KUKA KRL program: EPS_2_251191_MH01A_A_20251103013754.src

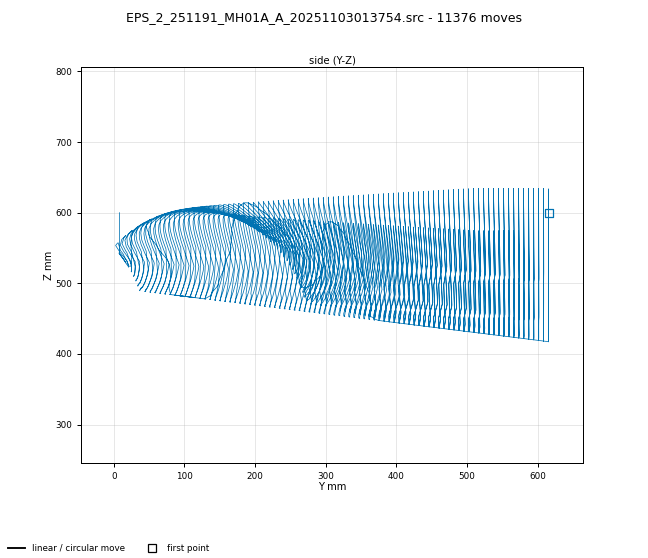
[picture p0: tool path of EPS_2_251191_MH01A_A_20251103013754.src, 11376 of 11378 moves have a stored position in this frame; points joined in program order, loops and branches not executed]
&ACCESS RVP
&REL 4
&COMMENT QRS 19112012
&PARAM EDITMASK = *
DEF PART()
EXT BAS (BAS_COMMAND :IN,REAL :IN )
INT I
BAS (#INITMOV,0 )

;KUKA QRS Post kuka4.cps  Date:22-06-2017 !

File_ID=2898

QRS_PRE_INIT()

;Init var - Until changes are made in qrs_pre_init
Outlet_Square_prg=0
Inlet_1_Square_prg=0
Inlet_2_Square_prg=0
Inlet_3_Square_prg=0
Inlet_4_Square_prg=0
Inlet_5_Square_prg=0

Outlet_1={X 0.000, Y 509.470, Z 509.000, B 0.000, E1 0.000 }
Inlet_1={X 0.000, Y 513.890, Z 449.000, B 0.000, E1 252.000 }
Outlet_1_type=251
Inlet_1_type=251
;QRS#1=Sidecore dimensions
;QRS#2=250-10" PVC SDR 35
;QRS#3=250-10" PVC SDR 35
;QRS#4=
;QRS#5=
;QRS#6=
;QRS#7=
;QRS#8=
;QRS#9=14M PSX
;QRS#10=14M PSX
;QRS#11=
;QRS#12=
;QRS#13=
;QRS#14=
;QRS#15=
;QRS#16=1220x127x914 3'
;QRS#17=EPS Height
;QRS#18=634,5
;QRS#19=*
;QRS#20= UPDATED VERSION 22-06-2017
;QRS#21=*
Outlet_Square=0100
Inlet_1_Square=0100
Inlet_2_Square=0
Inlet_3_Square=0
Inlet_4_Square=0
Inlet_5_Square=0
Mill_Square=1
Outlet_Square_Prg=205
Inlet_1_Square_prg=205

QRS_INIT()

$ADVANCE=5

; T1
PTP {E1 173.596,E2 173.596}
PTP {X 0,Y 615.507,A -85,B 0,C 180,E1 173.596,E2 173.596,E3 0,E4 0,E5 0,E6 0}
QRS_SPEED_INIT()
LIN {X 0,Y 615.507,Z 600,A -85,B 0,C 180,E1 173.596,E2 173.596,E3 0,E4 0,E5 0,E6 0} C_VEL
LIN {X 0,Y 615.507,Z 427.495,A -85,B 0,C 180,E1 173.596,E2 173.596} C_VEL
LIN {X 0,Y 615.507,Z 419.317,A -85,B 0,C 180,E1 173.596,E2 173.596} C_VEL
LIN {X 0,Y 615.493,Z 417.317,A -85,B 0,C 180,E1 173.409,E2 173.409} C_VEL
LIN {X 0,Y 615.481,Z 417.32,A -85,B 0,C 180,E1 170.801,E2 170.801} C_VEL
LIN {X 0,Y 615.475,Z 417.322,A -85,B 0,C 180,E1 168.139,E2 168.139} C_VEL
LIN {X 0,Y 615.49,Z 417.319,A -85,B 0,C 180,E1 165.451,E2 165.451} C_VEL
LIN {X 0,Y 615.49,Z 417.319,A -85,B 0,C 180,E1 162.729,E2 162.729} C_VEL
LIN {X 0,Y 615.486,Z 417.32,A -85,B 0,C 180,E1 159.967,E2 159.967} C_VEL
LIN {X 0,Y 615.477,Z 417.321,A -85,B 0,C 180,E1 157.155,E2 157.155} C_VEL
LIN {X 0,Y 615.484,Z 417.32,A -85,B 0,C 180,E1 154.43,E2 154.43} C_VEL
LIN {X 0,Y 615.492,Z 417.317,A -85,B 0,C 180,E1 151.547,E2 151.547} C_VEL
LIN {X 0,Y 615.483,Z 417.32,A -85,B 0,C 180,E1 148.913,E2 148.913} C_VEL
LIN {X 0,Y 615.486,Z 417.323,A -85,B 0,C 180,E1 146.465,E2 146.465} C_VEL
LIN {X 0,Y 615.488,Z 417.32,A -85,B 0,C 180,E1 143.575,E2 143.575} C_VEL
LIN {X 0,Y 615.484,Z 417.323,A -85,B 0,C 180,E1 140.937,E2 140.937} C_VEL
LIN {X 0,Y 615.487,Z 417.325,A -85,B 0,C 180,E1 138.526,E2 138.526} C_VEL
LIN {X 0,Y 615.491,Z 417.323,A -85,B 0,C 180,E1 135.85,E2 135.85} C_VEL
LIN {X 0,Y 615.492,Z 417.324,A -85,B 0,C 180,E1 133.047,E2 133.047} C_VEL
LIN {X 0,Y 615.497,Z 417.323,A -85,B 0,C 180,E1 130.09,E2 130.09} C_VEL
LIN {X 0,Y 615.484,Z 417.324,A -85,B 0,C 180,E1 127.242,E2 127.242} C_VEL
LIN {X 0,Y 615.496,Z 417.325,A -85,B 0,C 180,E1 124.701,E2 124.701} C_VEL
LIN {X 0,Y 615.48,Z 417.321,A -85,B 0,C 180,E1 122.329,E2 122.329} C_VEL
LIN {X 0,Y 615.498,Z 417.316,A -85,B 0,C 180,E1 119.796,E2 119.796} C_VEL
LIN {X 0,Y 615.486,Z 417.318,A -85,B 0,C 180,E1 117.044,E2 117.044} C_VEL
LIN {X 0,Y 615.478,Z 417.32,A -85,B 0,C 180,E1 114.272,E2 114.272} C_VEL
LIN {X 0,Y 615.479,Z 417.321,A -85,B 0,C 180,E1 111.432,E2 111.432} C_VEL
LIN {X 0,Y 615.481,Z 417.321,A -85,B 0,C 180,E1 108.602,E2 108.602} C_VEL
LIN {X 0,Y 615.491,Z 417.318,A -85,B 0,C 180,E1 105.905,E2 105.905} C_VEL
LIN {X 0,Y 615.48,Z 417.32,A -85,B 0,C 180,E1 103.201,E2 103.201} C_VEL
LIN {X 0,Y 615.478,Z 417.32,A -85,B 0,C 180,E1 100.527,E2 100.527} C_VEL
LIN {X 0,Y 615.489,Z 417.317,A -85,B 0,C 180,E1 97.875,E2 97.875} C_VEL
LIN {X 0,Y 615.484,Z 417.319,A -85,B 0,C 180,E1 95.241,E2 95.241} C_VEL
LIN {X 0,Y 615.478,Z 417.321,A -85,B 0,C 180,E1 92.618,E2 92.618} C_VEL
LIN {X 0,Y 615.491,Z 417.32,A -85,B 0,C 180,E1 90,E2 90} C_VEL
LIN {X 0,Y 615.484,Z 417.324,A -85,B 0,C 180,E1 87.382,E2 87.382} C_VEL
LIN {X 0,Y 615.493,Z 417.325,A -85,B 0,C 180,E1 84.759,E2 84.759} C_VEL
LIN {X 0,Y 615.487,Z 417.327,A -85,B 0,C 180,E1 82.125,E2 82.125} C_VEL
LIN {X 0,Y 615.488,Z 417.324,A -85,B 0,C 180,E1 79.473,E2 79.473} C_VEL
LIN {X 0,Y 615.482,Z 417.324,A -85,B 0,C 180,E1 76.799,E2 76.799} C_VEL
LIN {X 0,Y 615.491,Z 417.321,A -85,B 0,C 180,E1 74.095,E2 74.095} C_VEL
LIN {X 0,Y 615.483,Z 417.323,A -85,B 0,C 180,E1 71.354,E2 71.354} C_VEL
LIN {X 0,Y 615.482,Z 417.324,A -85,B 0,C 180,E1 68.568,E2 68.568} C_VEL
LIN {X 0,Y 615.495,Z 417.323,A -85,B 0,C 180,E1 65.729,E2 65.729} C_VEL
LIN {X 0,Y 615.486,Z 417.328,A -85,B 0,C 180,E1 62.823,E2 62.823} C_VEL
LIN {X 0,Y 615.497,Z 417.323,A -85,B 0,C 180,E1 60.205,E2 60.205} C_VEL
LIN {X 0,Y 615.488,Z 417.323,A -85,B 0,C 180,E1 57.543,E2 57.543} C_VEL
LIN {X 0,Y 615.496,Z 417.434,A -85,B 0,C 180,E1 55.979,E2 55.979} C_VEL
LIN {X 0,Y 615.483,Z 420.003,A -85,B 0,C 180,E1 53.576,E2 53.576} C_VEL
LIN {X 0,Y 615.485,Z 422.805,A -85,B 0,C 180,E1 50.939,E2 50.939} C_VEL
LIN {X 0,Y 615.495,Z 425.526,A -85,B 0,C 180,E1 48.528,E2 48.528} C_VEL
LIN {X 0,Y 615.478,Z 428.644,A -85,B 0,C 180,E1 45.851,E2 45.851} C_VEL
LIN {X 0,Y 615.493,Z 431.993,A -85,B 0,C 180,E1 43.049,E2 43.049} C_VEL
LIN {X 0,Y 615.486,Z 435.606,A -85,B 0,C 180,E1 40.09,E2 40.09} C_VEL
LIN {X 0,Y 615.491,Z 439.16,A -85,B 0,C 180,E1 37.242,E2 37.242} C_VEL
LIN {X 0,Y 615.478,Z 442.382,A -85,B 0,C 180,E1 34.701,E2 34.701} C_VEL
LIN {X 0,Y 615.494,Z 445.903,A -85,B 0,C 180,E1 31.968,E2 31.968} C_VEL
LIN {X 0,Y 615.485,Z 463.146,A -85,B 0,C 180,E1 31.611,E2 31.611} C_VEL
LIN {X 0,Y 615.49,Z 476.555,A -85,B 0,C 180,E1 31.199,E2 31.199} C_VEL
LIN {X 0,Y 615.481,Z 490.214,A -85,B 0,C 180,E1 30.635,E2 30.635} C_VEL
LIN {X 0,Y 615.495,Z 502.663,A -85,B 0,C 180,E1 29.979,E2 29.979} C_VEL
LIN {X 0,Y 615.497,Z 514.361,A -85,B 0,C 180,E1 29.218,E2 29.218} C_VEL
LIN {X 0,Y 615.499,Z 525.706,A -85,B 0,C 180,E1 28.319,E2 28.319} C_VEL
LIN {X 0,Y 615.496,Z 535.683,A -85,B 0,C 180,E1 27.361,E2 27.361} C_VEL
LIN {X 0,Y 615.499,Z 545.095,A -85,B 0,C 180,E1 26.261,E2 26.261} C_VEL
LIN {X 0,Y 615.497,Z 552.03,A -85,B 0,C 180,E1 25.282,E2 25.282} C_VEL
LIN {X 0,Y 615.495,Z 559.298,A -85,B 0,C 180,E1 24.012,E2 24.012} C_VEL
LIN {X 0,Y 615.494,Z 564.544,A -85,B 0,C 180,E1 22.844,E2 22.844} C_VEL
LIN {X 0,Y 615.493,Z 568.222,A -85,B 0,C 180,E1 21.784,E2 21.784} C_VEL
LIN {X 0,Y 615.495,Z 571.277,A -85,B 0,C 180,E1 20.561,E2 20.561} C_VEL
LIN {X 0,Y 615.494,Z 573.139,A -85,B 0,C 180,E1 19.338,E2 19.338} C_VEL
LIN {X 0,Y 615.497,Z 573.888,A -85,B 0,C 180,E1 17.957,E2 17.957} C_VEL
LIN {X 0,Y 615.493,Z 573.157,A -85,B 0,C 180,E1 16.587,E2 16.587} C_VEL
LIN {X 0,Y 615.492,Z 571.011,A -85,B 0,C 180,E1 15.226,E2 15.226} C_VEL
LIN {X 0,Y 615.496,Z 567.413,A -85,B 0,C 180,E1 13.874,E2 13.874} C_VEL
LIN {X 0,Y 615.496,Z 562.292,A -85,B 0,C 180,E1 12.53,E2 12.53} C_VEL
LIN {X 0,Y 615.496,Z 557.33,A -85,B 0,C 180,E1 11.527,E2 11.527} C_VEL
LIN {X 0,Y 615.498,Z 550.223,A -85,B 0,C 180,E1 10.361,E2 10.361} C_VEL
LIN {X 0,Y 615.496,Z 541.46,A -85,B 0,C 180,E1 9.199,E2 9.199} C_VEL
LIN {X 0,Y 615.497,Z 532.336,A -85,B 0,C 180,E1 8.206,E2 8.206} C_VEL
LIN {X 0,Y 615.496,Z 522.296,A -85,B 0,C 180,E1 7.298,E2 7.298} C_VEL
LIN {X 0,Y 615.5,Z 511.293,A -85,B 0,C 180,E1 6.474,E2 6.474} C_VEL
LIN {X 0,Y 615.486,Z 499.23,A -85,B 0,C 180,E1 5.734,E2 5.734} C_VEL
LIN {X 0,Y 615.478,Z 485.806,A -85,B 0,C 180,E1 5.077,E2 5.077} C_VEL
LIN {X 0,Y 615.489,Z 471.539,A -85,B 0,C 180,E1 4.544,E2 4.544} C_VEL
LIN {X 0,Y 615.493,Z 457.863,A -85,B 0,C 180,E1 4.175,E2 4.175} C_VEL
LIN {X 0,Y 615.487,Z 445.914,A -85,B 0,C 180,E1 3.949,E2 3.949} C_VEL
LIN {X 0,Y 615.486,Z 442.508,A -85,B 0,C 180,E1 1.309,E2 1.309} C_VEL
LIN {X 0,Y 615.486,Z 439.19,A -85,B 0,C 180,E1 -1.308,E2 -1.308} C_VEL
LIN {X 0,Y 615.477,Z 435.925,A -85,B 0,C 180,E1 -3.928,E2 -3.928} C_VEL
LIN {X 0,Y 615.49,Z 432.652,A -85,B 0,C 180,E1 -6.589,E2 -6.589} C_VEL
LIN {X 0,Y 615.494,Z 429.53,A -85,B 0,C 180,E1 -9.199,E2 -9.199} C_VEL
LIN {X 0,Y 615.477,Z 426.399,A -85,B 0,C 180,E1 -11.861,E2 -11.861} C_VEL
LIN {X 0,Y 615.493,Z 423.33,A -85,B 0,C 180,E1 -14.549,E2 -14.549} C_VEL
LIN {X 0,Y 615.49,Z 420.59,A -85,B 0,C 180,E1 -17.27,E2 -17.27} C_VEL
LIN {X 0,Y 615.488,Z 417.667,A -85,B 0,C 180,E1 -20.033,E2 -20.033} C_VEL
LIN {X 0,Y 615.479,Z 417.314,A -85,B 0,C 180,E1 -20.731,E2 -20.731} C_VEL
LIN {X 0,Y 615.489,Z 417.31,A -85,B 0,C 180,E1 -23.556,E2 -23.556} C_VEL
LIN {X 0,Y 615.493,Z 417.316,A -85,B 0,C 180,E1 -26.444,E2 -26.444} C_VEL
LIN {X 0,Y 615.48,Z 417.313,A -85,B 0,C 180,E1 -28.658,E2 -28.658} C_VEL
LIN {X 0,Y 615.483,Z 417.308,A -85,B 0,C 180,E1 -31.087,E2 -31.087} C_VEL
LIN {X 0,Y 615.489,Z 417.312,A -85,B 0,C 180,E1 -33.536,E2 -33.536} C_VEL
LIN {X 0,Y 615.488,Z 417.314,A -85,B 0,C 180,E1 -36.425,E2 -36.425} C_VEL
LIN {X 0,Y 615.482,Z 417.309,A -85,B 0,C 180,E1 -39.063,E2 -39.063} C_VEL
LIN {X 0,Y 615.492,Z 417.313,A -85,B 0,C 180,E1 -41.474,E2 -41.474} C_VEL
LIN {X 0,Y 615.493,Z 417.317,A -85,B 0,C 180,E1 -44.149,E2 -44.149} C_VEL
LIN {X 0,Y 615.481,Z 417.309,A -85,B 0,C 180,E1 -46.953,E2 -46.953} C_VEL
LIN {X 0,Y 615.489,Z 417.314,A -85,B 0,C 180,E1 -49.395,E2 -49.395} C_VEL
LIN {X 0,Y 615.49,Z 417.463,A -85,B 0,C 180,E1 -51.516,E2 -51.516} C_VEL
LIN {X 0,Y 615.491,Z 425.389,A -85,B 0,C 180,E1 -54.166,E2 -54.166} C_VEL
LIN {X 0,Y 615.495,Z 433.769,A -85,B 0,C 180,E1 -56.765,E2 -56.765} C_VEL
LIN {X 0,Y 615.477,Z 442.717,A -85,B 0,C 180,E1 -59.461,E2 -59.461} C_VEL
LIN {X 0,Y 615.491,Z 451.651,A -85,B 0,C 180,E1 -62.086,E2 -62.086} C_VEL
LIN {X 0,Y 615.477,Z 460.85,A -85,B 0,C 180,E1 -64.721,E2 -64.721} C_VEL
LIN {X 0,Y 615.493,Z 469.512,A -85,B 0,C 180,E1 -67.156,E2 -67.156} C_VEL
LIN {X 0,Y 615.485,Z 479.714,A -85,B 0,C 180,E1 -69.968,E2 -69.968} C_VEL
LIN {X 0,Y 615.499,Z 489.898,A -85,B 0,C 180,E1 -72.73,E2 -72.73} C_VEL
LIN {X 0,Y 615.479,Z 500.095,A -85,B 0,C 180,E1 -75.451,E2 -75.451} C_VEL
LIN {X 0,Y 615.49,Z 501.962,A -85,B 0,C 180,E1 -75.949,E2 -75.949} C_VEL
LIN {X 0,Y 615.492,Z 515.59,A -85,B 0,C 180,E1 -76.168,E2 -76.168} C_VEL
LIN {X 0,Y 615.487,Z 528.928,A -85,B 0,C 180,E1 -76.505,E2 -76.505} C_VEL
LIN {X 0,Y 615.492,Z 542.151,A -85,B 0,C 180,E1 -76.967,E2 -76.967} C_VEL
LIN {X 0,Y 615.478,Z 555.021,A -85,B 0,C 180,E1 -77.554,E2 -77.554} C_VEL
LIN {X 0,Y 615.497,Z 566.776,A -85,B 0,C 180,E1 -78.223,E2 -78.223} C_VEL
LIN {X 0,Y 615.496,Z 577.414,A -85,B 0,C 180,E1 -78.958,E2 -78.958} C_VEL
LIN {X 0,Y 615.498,Z 587.643,A -85,B 0,C 180,E1 -79.806,E2 -79.806} C_VEL
LIN {X 0,Y 615.498,Z 597.589,A -85,B 0,C 180,E1 -80.802,E2 -80.802} C_VEL
LIN {X 0,Y 615.496,Z 607.073,A -85,B 0,C 180,E1 -81.959,E2 -81.959} C_VEL
LIN {X 0,Y 615.495,Z 614.653,A -85,B 0,C 180,E1 -83.101,E2 -83.101} C_VEL
LIN {X 0,Y 615.494,Z 620.071,A -85,B 0,C 180,E1 -84.102,E2 -84.102} C_VEL
LIN {X 0,Y 615.495,Z 625.683,A -85,B 0,C 180,E1 -85.416,E2 -85.416} C_VEL
LIN {X 0,Y 615.495,Z 629.754,A -85,B 0,C 180,E1 -86.727,E2 -86.727} C_VEL
LIN {X 0,Y 615.497,Z 632.406,A -85,B 0,C 180,E1 -88.037,E2 -88.037} C_VEL
LIN {X 0,Y 615.493,Z 633.723,A -85,B 0,C 180,E1 -89.346,E2 -89.346} C_VEL
LIN {X 0,Y 615.493,Z 633.723,A -85,B 0,C 180,E1 -90.654,E2 -90.654} C_VEL
LIN {X 0,Y 615.497,Z 632.406,A -85,B 0,C 180,E1 -91.963,E2 -91.963} C_VEL
LIN {X 0,Y 615.495,Z 629.754,A -85,B 0,C 180,E1 -93.273,E2 -93.273} C_VEL
LIN {X 0,Y 615.495,Z 625.683,A -85,B 0,C 180,E1 -94.584,E2 -94.584} C_VEL
LIN {X 0,Y 615.494,Z 620.071,A -85,B 0,C 180,E1 -95.898,E2 -95.898} C_VEL
LIN {X 0,Y 615.495,Z 614.653,A -85,B 0,C 180,E1 -96.899,E2 -96.899} C_VEL
LIN {X 0,Y 615.496,Z 607.073,A -85,B 0,C 180,E1 -98.041,E2 -98.041} C_VEL
LIN {X 0,Y 615.498,Z 597.589,A -85,B 0,C 180,E1 -99.198,E2 -99.198} C_VEL
LIN {X 0,Y 615.498,Z 587.643,A -85,B 0,C 180,E1 -100.194,E2 -100.194} C_VEL
LIN {X 0,Y 615.498,Z 576.386,A -85,B 0,C 180,E1 -101.118,E2 -101.118} C_VEL
LIN {X 0,Y 615.496,Z 565.419,A -85,B 0,C 180,E1 -101.86,E2 -101.86} C_VEL
LIN {X 0,Y 615.479,Z 553.334,A -85,B 0,C 180,E1 -102.53,E2 -102.53} C_VEL
LIN {X 0,Y 615.488,Z 539.935,A -85,B 0,C 180,E1 -103.117,E2 -103.117} C_VEL
LIN {X 0,Y 615.488,Z 525.904,A -85,B 0,C 180,E1 -103.579,E2 -103.579} C_VEL
LIN {X 0,Y 615.496,Z 511.63,A -85,B 0,C 180,E1 -103.905,E2 -103.905} C_VEL
LIN {X 0,Y 615.49,Z 501.962,A -85,B 0,C 180,E1 -104.051,E2 -104.051} C_VEL
LIN {X 0,Y 615.494,Z 491.173,A -85,B 0,C 180,E1 -106.928,E2 -106.928} C_VEL
LIN {X 0,Y 615.486,Z 480.989,A -85,B 0,C 180,E1 -109.685,E2 -109.685} C_VEL
LIN {X 0,Y 615.481,Z 471.313,A -85,B 0,C 180,E1 -112.344,E2 -112.344} C_VEL
LIN {X 0,Y 615.488,Z 461.864,A -85,B 0,C 180,E1 -114.991,E2 -114.991} C_VEL
LIN {X 0,Y 615.481,Z 452.928,A -85,B 0,C 180,E1 -117.545,E2 -117.545} C_VEL
LIN {X 0,Y 615.476,Z 443.992,A -85,B 0,C 180,E1 -120.16,E2 -120.16} C_VEL
LIN {X 0,Y 615.489,Z 435.048,A -85,B 0,C 180,E1 -122.845,E2 -122.845} C_VEL
LIN {X 0,Y 615.491,Z 426.096,A -85,B 0,C 180,E1 -125.615,E2 -125.615} C_VEL
LIN {X 0,Y 615.49,Z 417.321,A -85,B 0,C 180,E1 -128.458,E2 -128.458} C_VEL
LIN {X 0,Y 615.487,Z 417.323,A -85,B 0,C 180,E1 -131.094,E2 -131.094} C_VEL
LIN {X 0,Y 615.482,Z 417.321,A -85,B 0,C 180,E1 -133.244,E2 -133.244} C_VEL
LIN {X 0,Y 615.485,Z 417.32,A -85,B 0,C 180,E1 -136.002,E2 -136.002} C_VEL
LIN {X 0,Y 615.494,Z 417.321,A -85,B 0,C 180,E1 -138.904,E2 -138.904} C_VEL
LIN {X 0,Y 615.491,Z 417.326,A -85,B 0,C 180,E1 -141.932,E2 -141.932} C_VEL
LIN {X 0,Y 615.48,Z 417.324,A -85,B 0,C 180,E1 -144.384,E2 -144.384} C_VEL
LIN {X 0,Y 615.492,Z 417.317,A -85,B 0,C 180,E1 -146.764,E2 -146.764} C_VEL
LIN {X 0,Y 615.481,Z 417.322,A -85,B 0,C 180,E1 -149.08,E2 -149.08} C_VEL
LIN {X 0,Y 615.492,Z 417.326,A -85,B 0,C 180,E1 -151.547,E2 -151.547} C_VEL
LIN {X 0,Y 615.497,Z 417.321,A -85,B 0,C 180,E1 -154.427,E2 -154.427} C_VEL
LIN {X 0,Y 615.482,Z 417.325,A -85,B 0,C 180,E1 -157.155,E2 -157.155} C_VEL
LIN {X 0,Y 615.487,Z 417.323,A -85,B 0,C 180,E1 -159.967,E2 -159.967} C_VEL
LIN {X 0,Y 615.489,Z 417.322,A -85,B 0,C 180,E1 -162.73,E2 -162.73} C_VEL
LIN {X 0,Y 615.495,Z 417.321,A -85,B 0,C 180,E1 -165.451,E2 -165.451} C_VEL
LIN {X 0,Y 615.493,Z 417.323,A -85,B 0,C 180,E1 -168.139,E2 -168.139} C_VEL
LIN {X 0,Y 615.494,Z 417.325,A -85,B 0,C 180,E1 -170.801,E2 -170.801} C_VEL
LIN {X 0,Y 615.495,Z 417.325,A -85,B 0,C 180,E1 -173.444,E2 -173.444} C_VEL
LIN {X 0,Y 615.486,Z 417.324,A -85,B 0,C 180,E1 -176.072,E2 -176.072} C_VEL
LIN {X 0,Y 615.495,Z 417.32,A -85,B 0,C 180,E1 -178.692,E2 -178.692} C_VEL
LIN {X 0,Y 615.486,Z 417.32,A -85,B 0,C 180,E1 -181.309,E2 -181.309} C_VEL
LIN {X 0,Y 615.476,Z 417.321,A -85,B 0,C 180,E1 -183.929,E2 -183.929} C_VEL
LIN {X 0,Y 615.493,Z 417.317,A -85,B 0,C 180,E1 -186.591,E2 -186.591} C_VEL
LIN {X 0,Y 614.815,Z 417.47,A -85,B 0,C 180,E1 -187.137,E2 -187.137} C_VEL
LIN {X 0,Y 611.974,Z 417.88,A -85,B 0,C 180,E1 -188.023,E2 -188.023} C_VEL
LIN {X 0,Y 609.578,Z 418.188,A -85,B 0,C 180,E1 -188.735,E2 -188.735} C_VEL
LIN {X 0,Y 608.543,Z 418.308,A -85,B 0,C 180,E1 -189.285,E2 -189.285} C_VEL
LIN {X 0,Y 608.455,Z 418.318,A -85,B 0,C 180,E1 -189.471,E2 -189.471} C_VEL
LIN {X 0,Y 608.454,Z 418.318,A -85,B 0,C 180,E1 -192,E2 -192} C_VEL
LIN {X 0,Y 608.476,Z 418.315,A -85,B 0,C 180,E1 -194.721,E2 -194.721} C_VEL
LIN {X 0,Y 608.452,Z 418.318,A -85,B 0,C 180,E1 -197.477,E2 -197.477} C_VEL
LIN {X 0,Y 608.465,Z 418.316,A -85,B 0,C 180,E1 -200.274,E2 -200.274} C_VEL
LIN {X 0,Y 608.454,Z 418.321,A -85,B 0,C 180,E1 -202.477,E2 -202.477} C_VEL
LIN {X 0,Y 608.459,Z 418.318,A -85,B 0,C 180,E1 -204.571,E2 -204.571} C_VEL
LIN {X 0,Y 608.474,Z 418.315,A -85,B 0,C 180,E1 -207.208,E2 -207.208} C_VEL
LIN {X 0,Y 608.46,Z 418.317,A -85,B 0,C 180,E1 -209.972,E2 -209.972} C_VEL
LIN {X 0,Y 608.463,Z 418.317,A -85,B 0,C 180,E1 -212.524,E2 -212.524} C_VEL
LIN {X 0,Y 608.44,Z 418.32,A -85,B 0,C 180,E1 -215.278,E2 -215.278} C_VEL
LIN {X 0,Y 608.47,Z 418.318,A -85,B 0,C 180,E1 -217.746,E2 -217.746} C_VEL
LIN {X 0,Y 608.449,Z 418.322,A -85,B 0,C 180,E1 -220.33,E2 -220.33} C_VEL
LIN {X 0,Y 608.463,Z 418.322,A -85,B 0,C 180,E1 -222.959,E2 -222.959} C_VEL
LIN {X 0,Y 608.461,Z 418.322,A -85,B 0,C 180,E1 -225.736,E2 -225.736} C_VEL
LIN {X 0,Y 608.461,Z 418.32,A -85,B 0,C 180,E1 -228.658,E2 -228.658} C_VEL
LIN {X 0,Y 608.469,Z 418.319,A -85,B 0,C 180,E1 -231.413,E2 -231.413} C_VEL
LIN {X 0,Y 608.479,Z 418.32,A -85,B 0,C 180,E1 -233.951,E2 -233.951} C_VEL
LIN {X 0,Y 608.469,Z 418.317,A -85,B 0,C 180,E1 -236.33,E2 -236.33} C_VEL
LIN {X 0,Y 608.447,Z 418.319,A -85,B 0,C 180,E1 -238.733,E2 -238.733} C_VEL
LIN {X 0,Y 608.469,Z 418.316,A -85,B 0,C 180,E1 -241.381,E2 -241.381} C_VEL
LIN {X 0,Y 608.475,Z 418.315,A -85,B 0,C 180,E1 -244.279,E2 -244.279} C_VEL
LIN {X 0,Y 608.451,Z 418.318,A -85,B 0,C 180,E1 -246.876,E2 -246.876} C_VEL
LIN {X 0,Y 608.464,Z 418.319,A -85,B 0,C 180,E1 -249.323,E2 -249.323} C_VEL
LIN {X 0,Y 608.456,Z 418.323,A -85,B 0,C 180,E1 -251.829,E2 -251.829} C_VEL
LIN {X 0,Y 608.473,Z 418.32,A -85,B 0,C 180,E1 -254.594,E2 -254.594} C_VEL
LIN {X 0,Y 608.478,Z 418.32,A -85,B 0,C 180,E1 -257.323,E2 -257.323} C_VEL
LIN {X 0,Y 608.459,Z 418.322,A -85,B 0,C 180,E1 -260.023,E2 -260.023} C_VEL
LIN {X 0,Y 608.467,Z 418.32,A -85,B 0,C 180,E1 -262.701,E2 -262.701} C_VEL
LIN {X 0,Y 608.452,Z 418.321,A -85,B 0,C 180,E1 -265.362,E2 -265.362} C_VEL
LIN {X 0,Y 608.468,Z 418.318,A -85,B 0,C 180,E1 -268.014,E2 -268.014} C_VEL
LIN {X 0,Y 608.472,Z 418.317,A -85,B 0,C 180,E1 -270.662,E2 -270.662} C_VEL
LIN {X 0,Y 608.476,Z 418.316,A -85,B 0,C 180,E1 -273.311,E2 -273.311} C_VEL
LIN {X 0,Y 608.468,Z 418.316,A -85,B 0,C 180,E1 -275.967,E2 -275.967} C_VEL
LIN {X 0,Y 608.451,Z 418.318,A -85,B 0,C 180,E1 -278.636,E2 -278.636} C_VEL
LIN {X 0,Y 608.46,Z 418.317,A -85,B 0,C 180,E1 -281.324,E2 -281.324} C_VEL
LIN {X 0,Y 608.474,Z 418.315,A -85,B 0,C 180,E1 -284.037,E2 -284.037} C_VEL
LIN {X 0,Y 608.442,Z 418.319,A -85,B 0,C 180,E1 -286.784,E2 -286.784} C_VEL
LIN {X 0,Y 608.449,Z 418.319,A -85,B 0,C 180,E1 -289.57,E2 -289.57} C_VEL
LIN {X 0,Y 608.462,Z 418.317,A -85,B 0,C 180,E1 -292.476,E2 -292.476} C_VEL
LIN {X 0,Y 608.459,Z 418.32,A -85,B 0,C 180,E1 -294.57,E2 -294.57} C_VEL
LIN {X 0,Y 608.481,Z 418.319,A -85,B 0,C 180,E1 -297.207,E2 -297.207} C_VEL
LIN {X 0,Y 608.47,Z 418.32,A -85,B 0,C 180,E1 -299.971,E2 -299.971} C_VEL
LIN {X 0,Y 608.463,Z 418.32,A -85,B 0,C 180,E1 -302.522,E2 -302.522} C_VEL
LIN {X 0,Y 608.472,Z 418.317,A -85,B 0,C 180,E1 -303.734,E2 -303.734} C_VEL
LIN {X 0,Y 608.451,Z 419.606,A -85,B 0,C 180,E1 -305.276,E2 -305.276} C_VEL
LIN {X 0,Y 608.428,Z 422.745,A -85,B 0,C 180,E1 -308.235,E2 -308.235} C_VEL
LIN {X 0,Y 608.43,Z 424.998,A -85,B 0,C 180,E1 -310.326,E2 -310.326} C_VEL
LIN {X 0,Y 608.433,Z 428.416,A -85,B 0,C 180,E1 -313.305,E2 -313.305} C_VEL
LIN {X 0,Y 608.418,Z 431.745,A -85,B 0,C 180,E1 -316.126,E2 -316.126} C_VEL
LIN {X 0,Y 608.421,Z 434.805,A -85,B 0,C 180,E1 -318.661,E2 -318.661} C_VEL
LIN {X 0,Y 608.403,Z 438.187,A -85,B 0,C 180,E1 -321.407,E2 -321.407} C_VEL
LIN {X 0,Y 608.416,Z 441.382,A -85,B 0,C 180,E1 -323.957,E2 -323.957} C_VEL
LIN {X 0,Y 608.428,Z 444.393,A -85,B 0,C 180,E1 -326.327,E2 -326.327} C_VEL
LIN {X 0,Y 608.463,Z 446.533,A -85,B 0,C 180,E1 -327.892,E2 -327.892} C_VEL
LIN {X 0,Y 608.595,Z 461.114,A -85,B 0,C 180,E1 -328.181,E2 -328.181} C_VEL
LIN {X 0,Y 608.586,Z 475.036,A -85,B 0,C 180,E1 -328.593,E2 -328.593} C_VEL
LIN {X 0,Y 608.529,Z 488.243,A -85,B 0,C 180,E1 -329.121,E2 -329.121} C_VEL
LIN {X 0,Y 608.532,Z 501.009,A -85,B 0,C 180,E1 -329.777,E2 -329.777} C_VEL
LIN {X 0,Y 608.522,Z 512.531,A -85,B 0,C 180,E1 -330.509,E2 -330.509} C_VEL
LIN {X 0,Y 608.48,Z 523.778,A -85,B 0,C 180,E1 -331.377,E2 -331.377} C_VEL
LIN {X 0,Y 608.477,Z 533.667,A -85,B 0,C 180,E1 -332.296,E2 -332.296} C_VEL
LIN {X 0,Y 608.468,Z 543.576,A -85,B 0,C 180,E1 -333.412,E2 -333.412} C_VEL
LIN {X 0,Y 608.447,Z 551.446,A -85,B 0,C 180,E1 -334.49,E2 -334.49} C_VEL
LIN {X 0,Y 608.441,Z 558.485,A -85,B 0,C 180,E1 -335.675,E2 -335.675} C_VEL
LIN {X 0,Y 608.44,Z 564.134,A -85,B 0,C 180,E1 -336.875,E2 -336.875} C_VEL
LIN {X 0,Y 608.453,Z 568.059,A -85,B 0,C 180,E1 -337.951,E2 -337.951} C_VEL
LIN {X 0,Y 608.437,Z 571.679,A -85,B 0,C 180,E1 -339.326,E2 -339.326} C_VEL
LIN {X 0,Y 608.414,Z 573.485,A -85,B 0,C 180,E1 -340.428,E2 -340.428} C_VEL
LIN {X 0,Y 608.423,Z 574.455,A -85,B 0,C 180,E1 -341.827,E2 -341.827} C_VEL
LIN {X 0,Y 608.419,Z 573.974,A -85,B 0,C 180,E1 -343.215,E2 -343.215} C_VEL
LIN {X 0,Y 608.418,Z 572.048,A -85,B 0,C 180,E1 -344.592,E2 -344.592} C_VEL
LIN {X 0,Y 608.434,Z 568.526,A -85,B 0,C 180,E1 -345.992,E2 -345.992} C_VEL
LIN {X 0,Y 608.427,Z 563.676,A -85,B 0,C 180,E1 -347.322,E2 -347.322} C_VEL
LIN {X 0,Y 608.433,Z 558.905,A -85,B 0,C 180,E1 -348.338,E2 -348.338} C_VEL
LIN {X 0,Y 608.455,Z 551.993,A -85,B 0,C 180,E1 -349.518,E2 -349.518} C_VEL
LIN {X 0,Y 608.477,Z 544.81,A -85,B 0,C 180,E1 -350.526,E2 -350.526} C_VEL
LIN {X 0,Y 608.485,Z 536.206,A -85,B 0,C 180,E1 -351.532,E2 -351.532} C_VEL
LIN {X 0,Y 608.496,Z 525.838,A -85,B 0,C 180,E1 -352.534,E2 -352.534} C_VEL
LIN {X 0,Y 608.509,Z 515.477,A -85,B 0,C 180,E1 -353.368,E2 -353.368} C_VEL
LIN {X 0,Y 608.509,Z 502.901,A -85,B 0,C 180,E1 -354.2,E2 -354.2} C_VEL
LIN {X 0,Y 608.545,Z 490.403,A -85,B 0,C 180,E1 -354.865,E2 -354.865} C_VEL
LIN {X 0,Y 608.559,Z 477.572,A -85,B 0,C 180,E1 -355.404,E2 -355.404} C_VEL
LIN {X 0,Y 608.584,Z 463.812,A -85,B 0,C 180,E1 -355.84,E2 -355.84} C_VEL
LIN {X 0,Y 608.604,Z 449.456,A -85,B 0,C 180,E1 -356.151,E2 -356.151} C_VEL
LIN {X 0,Y 608.437,Z 446.383,A -85,B 0,C 180,E1 -356.212,E2 -356.212} C_VEL
LIN {X 0,Y 608.438,Z 443.228,A -85,B 0,C 180,E1 -358.676,E2 -358.676} C_VEL
LIN {X 0,Y 608.438,Z 439.883,A -85,B 0,C 180,E1 -361.324,E2 -361.324} C_VEL
LIN {X 0,Y 608.415,Z 436.589,A -85,B 0,C 180,E1 -363.974,E2 -363.974} C_VEL
LIN {X 0,Y 608.428,Z 433.344,A -85,B 0,C 180,E1 -366.633,E2 -366.633} C_VEL
LIN {X 0,Y 608.426,Z 430.15,A -85,B 0,C 180,E1 -369.306,E2 -369.306} C_VEL
LIN {X 0,Y 608.416,Z 427.01,A -85,B 0,C 180,E1 -372.001,E2 -372.001} C_VEL
LIN {X 0,Y 608.447,Z 424.007,A -85,B 0,C 180,E1 -374.721,E2 -374.721} C_VEL
LIN {X 0,Y 608.455,Z 421.256,A -85,B 0,C 180,E1 -377.476,E2 -377.476} C_VEL
LIN {X 0,Y 608.454,Z 419.052,A -85,B 0,C 180,E1 -379.57,E2 -379.57} C_VEL
LIN {X 0,Y 608.429,Z 418.326,A -85,B 0,C 180,E1 -380.275,E2 -380.275} C_VEL
LIN {X 0,Y 608.456,Z 418.318,A -85,B 0,C 180,E1 -382.478,E2 -382.478} C_VEL
LIN {X 0,Y 608.452,Z 418.317,A -85,B 0,C 180,E1 -384.571,E2 -384.571} C_VEL
LIN {X 0,Y 608.473,Z 418.31,A -85,B 0,C 180,E1 -387.208,E2 -387.208} C_VEL
LIN {X 0,Y 608.47,Z 418.319,A -85,B 0,C 180,E1 -389.974,E2 -389.974} C_VEL
LIN {X 0,Y 608.463,Z 418.314,A -85,B 0,C 180,E1 -392.524,E2 -392.524} C_VEL
LIN {X 0,Y 608.441,Z 418.315,A -85,B 0,C 180,E1 -395.278,E2 -395.278} C_VEL
LIN {X 0,Y 608.471,Z 418.317,A -85,B 0,C 180,E1 -397.746,E2 -397.746} C_VEL
LIN {X 0,Y 608.448,Z 418.317,A -85,B 0,C 180,E1 -400.33,E2 -400.33} C_VEL
LIN {X 0,Y 608.453,Z 418.313,A -85,B 0,C 180,E1 -402.96,E2 -402.96} C_VEL
LIN {X 0,Y 608.463,Z 418.32,A -85,B 0,C 180,E1 -405.736,E2 -405.736} C_VEL
LIN {X 0,Y 608.457,Z 418.313,A -85,B 0,C 180,E1 -408.658,E2 -408.658} C_VEL
LIN {X 0,Y 608.494,Z 418.458,A -85,B 0,C 180,E1 -411.309,E2 -411.309} C_VEL
LIN {X 0,Y 608.539,Z 424.801,A -85,B 0,C 180,E1 -413.504,E2 -413.504} C_VEL
LIN {X 0,Y 608.521,Z 432.421,A -85,B 0,C 180,E1 -415.935,E2 -415.935} C_VEL
LIN {X 0,Y 608.521,Z 441.58,A -85,B 0,C 180,E1 -418.721,E2 -418.721} C_VEL
LIN {X 0,Y 608.499,Z 450.481,A -85,B 0,C 180,E1 -421.376,E2 -421.376} C_VEL
LIN {X 0,Y 608.492,Z 460.46,A -85,B 0,C 180,E1 -424.275,E2 -424.275} C_VEL
LIN {X 0,Y 608.461,Z 469.627,A -85,B 0,C 180,E1 -426.877,E2 -426.877} C_VEL
LIN {X 0,Y 608.464,Z 478.403,A -85,B 0,C 180,E1 -429.322,E2 -429.322} C_VEL
LIN {X 0,Y 608.449,Z 488.826,A -85,B 0,C 180,E1 -432.176,E2 -432.176} C_VEL
LIN {X 0,Y 608.44,Z 499.066,A -85,B 0,C 180,E1 -434.937,E2 -434.937} C_VEL
LIN {X 0,Y 608.457,Z 502.3,A -85,B 0,C 180,E1 -435.788,E2 -435.788} C_VEL
LIN {X 0,Y 608.606,Z 516.831,A -85,B 0,C 180,E1 -436.036,E2 -436.036} C_VEL
LIN {X 0,Y 608.584,Z 530.267,A -85,B 0,C 180,E1 -436.391,E2 -436.391} C_VEL
LIN {X 0,Y 608.552,Z 542.177,A -85,B 0,C 180,E1 -436.816,E2 -436.816} C_VEL
LIN {X 0,Y 608.517,Z 555.076,A -85,B 0,C 180,E1 -437.409,E2 -437.409} C_VEL
LIN {X 0,Y 608.534,Z 568.15,A -85,B 0,C 180,E1 -438.171,E2 -438.171} C_VEL
LIN {X 0,Y 608.506,Z 580.042,A -85,B 0,C 180,E1 -439.027,E2 -439.027} C_VEL
LIN {X 0,Y 608.472,Z 591.392,A -85,B 0,C 180,E1 -440.023,E2 -440.023} C_VEL
LIN {X 0,Y 608.473,Z 600.824,A -85,B 0,C 180,E1 -441.03,E2 -441.03} C_VEL
LIN {X 0,Y 608.453,Z 609.798,A -85,B 0,C 180,E1 -442.2,E2 -442.2} C_VEL
LIN {X 0,Y 608.441,Z 617.227,A -85,B 0,C 180,E1 -443.399,E2 -443.399} C_VEL
LIN {X 0,Y 608.44,Z 623.568,A -85,B 0,C 180,E1 -444.698,E2 -444.698} C_VEL
LIN {X 0,Y 608.431,Z 628.441,A -85,B 0,C 180,E1 -446.026,E2 -446.026} C_VEL
LIN {X 0,Y 608.424,Z 631.831,A -85,B 0,C 180,E1 -447.352,E2 -447.352} C_VEL
LIN {X 0,Y 608.442,Z 633.83,A -85,B 0,C 180,E1 -448.676,E2 -448.676} C_VEL
LIN {X 0,Y 608.433,Z 634.5,A -85,B 0,C 180,E1 -450,E2 -450} C_VEL
LIN {X 0,Y 608.442,Z 633.83,A -85,B 0,C 180,E1 -451.324,E2 -451.324} C_VEL
LIN {X 0,Y 608.424,Z 631.831,A -85,B 0,C 180,E1 -452.648,E2 -452.648} C_VEL
LIN {X 0,Y 608.431,Z 628.441,A -85,B 0,C 180,E1 -453.974,E2 -453.974} C_VEL
LIN {X 0,Y 608.44,Z 623.568,A -85,B 0,C 180,E1 -455.302,E2 -455.302} C_VEL
LIN {X 0,Y 608.445,Z 617.212,A -85,B 0,C 180,E1 -456.603,E2 -456.603} C_VEL
LIN {X 0,Y 608.453,Z 609.798,A -85,B 0,C 180,E1 -457.8,E2 -457.8} C_VEL
LIN {X 0,Y 608.473,Z 600.824,A -85,B 0,C 180,E1 -458.97,E2 -458.97} C_VEL
LIN {X 0,Y 608.472,Z 591.392,A -85,B 0,C 180,E1 -459.977,E2 -459.977} C_VEL
LIN {X 0,Y 608.505,Z 580.048,A -85,B 0,C 180,E1 -460.973,E2 -460.973} C_VEL
LIN {X 0,Y 608.534,Z 568.15,A -85,B 0,C 180,E1 -461.829,E2 -461.829} C_VEL
LIN {X 0,Y 608.517,Z 555.076,A -85,B 0,C 180,E1 -462.591,E2 -462.591} C_VEL
LIN {X 0,Y 608.552,Z 542.177,A -85,B 0,C 180,E1 -463.184,E2 -463.184} C_VEL
LIN {X 0,Y 608.588,Z 528.188,A -85,B 0,C 180,E1 -463.672,E2 -463.672} C_VEL
LIN {X 0,Y 608.621,Z 514.464,A -85,B 0,C 180,E1 -464.012,E2 -464.012} C_VEL
LIN {X 0,Y 608.459,Z 502.241,A -85,B 0,C 180,E1 -464.215,E2 -464.215} C_VEL
LIN {X 0,Y 608.451,Z 492.666,A -85,B 0,C 180,E1 -466.784,E2 -466.784} C_VEL
LIN {X 0,Y 608.458,Z 482.426,A -85,B 0,C 180,E1 -469.57,E2 -469.57} C_VEL
LIN {X 0,Y 608.477,Z 472.187,A -85,B 0,C 180,E1 -472.405,E2 -472.405} C_VEL
LIN {X 0,Y 608.465,Z 461.947,A -85,B 0,C 180,E1 -475.3,E2 -475.3} C_VEL
LIN {X 0,Y 608.502,Z 452.987,A -85,B 0,C 180,E1 -477.889,E2 -477.889} C_VEL
LIN {X 0,Y 608.523,Z 442.804,A -85,B 0,C 180,E1 -480.909,E2 -480.909} C_VEL
LIN {X 0,Y 608.532,Z 433.502,A -85,B 0,C 180,E1 -483.743,E2 -483.743} C_VEL
LIN {X 0,Y 608.554,Z 424.821,A -85,B 0,C 180,E1 -486.495,E2 -486.495} C_VEL
LIN {X 0,Y 608.473,Z 418.317,A -85,B 0,C 180,E1 -488.666,E2 -488.666} C_VEL
LIN {X 0,Y 608.461,Z 418.318,A -85,B 0,C 180,E1 -491.342,E2 -491.342} C_VEL
LIN {X 0,Y 608.45,Z 418.319,A -85,B 0,C 180,E1 -494.263,E2 -494.263} C_VEL
LIN {X 0,Y 608.452,Z 418.318,A -85,B 0,C 180,E1 -497.04,E2 -497.04} C_VEL
LIN {X 0,Y 608.449,Z 418.319,A -85,B 0,C 180,E1 -499.696,E2 -499.696} C_VEL
LIN {X 0,Y 608.472,Z 418.317,A -85,B 0,C 180,E1 -502.254,E2 -502.254} C_VEL
LIN {X 0,Y 608.442,Z 418.32,A -85,B 0,C 180,E1 -505.094,E2 -505.094} C_VEL
LIN {X 0,Y 608.467,Z 418.32,A -85,B 0,C 180,E1 -507.475,E2 -507.475} C_VEL
LIN {X 0,Y 608.48,Z 418.319,A -85,B 0,C 180,E1 -510.221,E2 -510.221} C_VEL
LIN {X 0,Y 608.482,Z 418.318,A -85,B 0,C 180,E1 -512.79,E2 -512.79} C_VEL
LIN {X 0,Y 608.45,Z 418.321,A -85,B 0,C 180,E1 -515.429,E2 -515.429} C_VEL
LIN {X 0,Y 608.473,Z 418.32,A -85,B 0,C 180,E1 -518.309,E2 -518.309} C_VEL
LIN {X 0,Y 608.469,Z 418.319,A -85,B 0,C 180,E1 -521.281,E2 -521.281} C_VEL
LIN {X 0,Y 608.464,Z 418.322,A -85,B 0,C 180,E1 -523.906,E2 -523.906} C_VEL
LIN {X 0,Y 608.46,Z 418.322,A -85,B 0,C 180,E1 -526.644,E2 -526.644} C_VEL
LIN {X 0,Y 608.47,Z 418.321,A -85,B 0,C 180,E1 -529.35,E2 -529.35} C_VEL
LIN {X 0,Y 608.477,Z 418.319,A -85,B 0,C 180,E1 -532.033,E2 -532.033} C_VEL
LIN {X 0,Y 608.471,Z 418.319,A -85,B 0,C 180,E1 -534.698,E2 -534.698} C_VEL
LIN {X 0,Y 608.479,Z 418.317,A -85,B 0,C 180,E1 -537.352,E2 -537.352} C_VEL
LIN {X 0,Y 608.469,Z 418.317,A -85,B 0,C 180,E1 -540,E2 -540} C_VEL
LIN {X 0,Y 608.484,Z 418.315,A -85,B 0,C 180,E1 -542.648,E2 -542.648} C_VEL
LIN {X 0,Y 608.464,Z 418.317,A -85,B 0,C 180,E1 -545.302,E2 -545.302} C_VEL
LIN {X 0,Y 608.471,Z 418.316,A -85,B 0,C 180,E1 -547.967,E2 -547.967} C_VEL
LIN {X 0,Y 608.455,Z 418.318,A -85,B 0,C 180,E1 -549.471,E2 -549.471} C_VEL
LIN {X 0,Y 607.778,Z 418.407,A -85,B 0,C 180,E1 -550.024,E2 -550.024} C_VEL
LIN {X 0,Y 604.921,Z 418.759,A -85,B 0,C 180,E1 -550.921,E2 -550.921} C_VEL
LIN {X 0,Y 602.516,Z 419.059,A -85,B 0,C 180,E1 -551.642,E2 -551.642} C_VEL
LIN {X 0,Y 601.489,Z 419.186,A -85,B 0,C 180,E1 -552.199,E2 -552.199} C_VEL
LIN {X 0,Y 601.407,Z 419.196,A -85,B 0,C 180,E1 -552.387,E2 -552.387} C_VEL
LIN {X 0,Y 601.429,Z 419.193,A -85,B 0,C 180,E1 -554.897,E2 -554.897} C_VEL
LIN {X 0,Y 601.432,Z 419.196,A -85,B 0,C 180,E1 -556.986,E2 -556.986} C_VEL
LIN {X 0,Y 601.406,Z 419.198,A -85,B 0,C 180,E1 -559.81,E2 -559.81} C_VEL
LIN {X 0,Y 601.41,Z 419.197,A -85,B 0,C 180,E1 -562.606,E2 -562.606} C_VEL
LIN {X 0,Y 601.405,Z 419.199,A -85,B 0,C 180,E1 -564.879,E2 -564.879} C_VEL
LIN {X 0,Y 601.422,Z 419.199,A -85,B 0,C 180,E1 -567.868,E2 -567.868} C_VEL
LIN {X 0,Y 601.423,Z 419.195,A -85,B 0,C 180,E1 -570.165,E2 -570.165} C_VEL
LIN {X 0,Y 601.424,Z 419.194,A -85,B 0,C 180,E1 -572.717,E2 -572.717} C_VEL
LIN {X 0,Y 601.397,Z 419.198,A -85,B 0,C 180,E1 -575.114,E2 -575.114} C_VEL
LIN {X 0,Y 601.433,Z 419.197,A -85,B 0,C 180,E1 -577.42,E2 -577.42} C_VEL
LIN {X 0,Y 601.399,Z 419.199,A -85,B 0,C 180,E1 -579.996,E2 -579.996} C_VEL
LIN {X 0,Y 601.438,Z 419.194,A -85,B 0,C 180,E1 -582.668,E2 -582.668} C_VEL
LIN {X 0,Y 601.424,Z 419.196,A -85,B 0,C 180,E1 -585.483,E2 -585.483} C_VEL
LIN {X 0,Y 601.422,Z 419.199,A -85,B 0,C 180,E1 -588.408,E2 -588.408} C_VEL
LIN {X 0,Y 601.435,Z 419.194,A -85,B 0,C 180,E1 -590.876,E2 -590.876} C_VEL
LIN {X 0,Y 601.443,Z 419.194,A -85,B 0,C 180,E1 -593.735,E2 -593.735} C_VEL
LIN {X 0,Y 601.436,Z 419.192,A -85,B 0,C 180,E1 -596.064,E2 -596.064} C_VEL
LIN {X 0,Y 601.421,Z 419.194,A -85,B 0,C 180,E1 -598.546,E2 -598.546} C_VEL
LIN {X 0,Y 601.437,Z 419.193,A -85,B 0,C 180,E1 -601.212,E2 -601.212} C_VEL
LIN {X 0,Y 601.408,Z 419.2,A -85,B 0,C 180,E1 -603.637,E2 -603.637} C_VEL
LIN {X 0,Y 601.421,Z 419.196,A -85,B 0,C 180,E1 -606.59,E2 -606.59} C_VEL
LIN {X 0,Y 601.429,Z 419.194,A -85,B 0,C 180,E1 -609.479,E2 -609.479} C_VEL
LIN {X 0,Y 601.398,Z 419.197,A -85,B 0,C 180,E1 -612.312,E2 -612.312} C_VEL
LIN {X 0,Y 601.417,Z 419.198,A -85,B 0,C 180,E1 -614.409,E2 -614.409} C_VEL
LIN {X 0,Y 601.422,Z 419.197,A -85,B 0,C 180,E1 -617.172,E2 -617.172} C_VEL
LIN {X 0,Y 601.435,Z 419.196,A -85,B 0,C 180,E1 -619.905,E2 -619.905} C_VEL
LIN {X 0,Y 601.445,Z 419.194,A -85,B 0,C 180,E1 -622.615,E2 -622.615} C_VEL
LIN {X 0,Y 601.421,Z 419.196,A -85,B 0,C 180,E1 -625.308,E2 -625.308} C_VEL
LIN {X 0,Y 601.437,Z 419.194,A -85,B 0,C 180,E1 -627.991,E2 -627.991} C_VEL
LIN {X 0,Y 601.444,Z 419.192,A -85,B 0,C 180,E1 -630.67,E2 -630.67} C_VEL
LIN {X 0,Y 601.428,Z 419.194,A -85,B 0,C 180,E1 -633.35,E2 -633.35} C_VEL
LIN {X 0,Y 601.421,Z 419.194,A -85,B 0,C 180,E1 -636.037,E2 -636.037} C_VEL
LIN {X 0,Y 601.414,Z 419.195,A -85,B 0,C 180,E1 -638.738,E2 -638.738} C_VEL
LIN {X 0,Y 601.427,Z 419.193,A -85,B 0,C 180,E1 -641.458,E2 -641.458} C_VEL
LIN {X 0,Y 601.424,Z 419.194,A -85,B 0,C 180,E1 -644.205,E2 -644.205} C_VEL
LIN {X 0,Y 601.415,Z 419.195,A -85,B 0,C 180,E1 -646.986,E2 -646.986} C_VEL
LIN {X 0,Y 601.406,Z 419.196,A -85,B 0,C 180,E1 -649.809,E2 -649.809} C_VEL
LIN {X 0,Y 601.415,Z 419.196,A -85,B 0,C 180,E1 -652.682,E2 -652.682} C_VEL
LIN {X 0,Y 601.405,Z 419.197,A -85,B 0,C 180,E1 -654.878,E2 -654.878} C_VEL
LIN {X 0,Y 601.425,Z 419.193,A -85,B 0,C 180,E1 -657.867,E2 -657.867} C_VEL
LIN {X 0,Y 601.43,Z 419.195,A -85,B 0,C 180,E1 -660.163,E2 -660.163} C_VEL
LIN {X 0,Y 601.422,Z 419.198,A -85,B 0,C 180,E1 -662.715,E2 -662.715} C_VEL
LIN {X 0,Y 601.385,Z 419.203,A -85,B 0,C 180,E1 -664.12,E2 -664.12} C_VEL
LIN {X 0,Y 601.358,Z 421.213,A -85,B 0,C 180,E1 -666.254,E2 -666.254} C_VEL
LIN {X 0,Y 601.357,Z 424.247,A -85,B 0,C 180,E1 -669.13,E2 -669.13} C_VEL
LIN {X 0,Y 601.342,Z 427.09,A -85,B 0,C 180,E1 -671.771,E2 -671.771} C_VEL
LIN {X 0,Y 601.36,Z 430.258,A -85,B 0,C 180,E1 -674.528,E2 -674.528} C_VEL
LIN {X 0,Y 601.377,Z 433.657,A -85,B 0,C 180,E1 -677.412,E2 -677.412} C_VEL
LIN {X 0,Y 601.313,Z 437.362,A -85,B 0,C 180,E1 -680.478,E2 -680.478} C_VEL
LIN {X 0,Y 601.325,Z 440.009,A -85,B 0,C 180,E1 -682.63,E2 -682.63} C_VEL
LIN {X 0,Y 601.34,Z 443.041,A -85,B 0,C 180,E1 -685.063,E2 -685.063} C_VEL
LIN {X 0,Y 601.363,Z 446.393,A -85,B 0,C 180,E1 -687.715,E2 -687.715} C_VEL
LIN {X 0,Y 601.726,Z 452.076,A -85,B 0,C 180,E1 -687.824,E2 -687.824} C_VEL
LIN {X 0,Y 601.667,Z 466.537,A -85,B 0,C 180,E1 -688.165,E2 -688.165} C_VEL
LIN {X 0,Y 601.661,Z 479.264,A -85,B 0,C 180,E1 -688.594,E2 -688.594} C_VEL
LIN {X 0,Y 601.601,Z 492.456,A -85,B 0,C 180,E1 -689.175,E2 -689.175} C_VEL
LIN {X 0,Y 601.546,Z 505.474,A -85,B 0,C 180,E1 -689.903,E2 -689.903} C_VEL
LIN {X 0,Y 601.51,Z 516.917,A -85,B 0,C 180,E1 -690.695,E2 -690.695} C_VEL
LIN {X 0,Y 601.453,Z 528.356,A -85,B 0,C 180,E1 -691.66,E2 -691.66} C_VEL
LIN {X 0,Y 601.422,Z 538.473,A -85,B 0,C 180,E1 -692.7,E2 -692.7} C_VEL
LIN {X 0,Y 601.406,Z 547.132,A -85,B 0,C 180,E1 -693.777,E2 -693.777} C_VEL
LIN {X 0,Y 601.385,Z 554.771,A -85,B 0,C 180,E1 -694.936,E2 -694.936} C_VEL
LIN {X 0,Y 601.375,Z 561.557,A -85,B 0,C 180,E1 -696.222,E2 -696.222} C_VEL
LIN {X 0,Y 601.374,Z 566.38,A -85,B 0,C 180,E1 -697.402,E2 -697.402} C_VEL
LIN {X 0,Y 601.32,Z 570.48,A -85,B 0,C 180,E1 -698.757,E2 -698.757} C_VEL
LIN {X 0,Y 601.349,Z 572.063,A -85,B 0,C 180,E1 -699.475,E2 -699.475} C_VEL
LIN {X 0,Y 601.311,Z 574,A -85,B 0,C 180,E1 -700.897,E2 -700.897} C_VEL
LIN {X 0,Y 601.309,Z 574.445,A -85,B 0,C 180,E1 -702.309,E2 -702.309} C_VEL
LIN {X 0,Y 601.345,Z 573.451,A -85,B 0,C 180,E1 -703.71,E2 -703.71} C_VEL
LIN {X 0,Y 601.316,Z 571.029,A -85,B 0,C 180,E1 -705.1,E2 -705.1} C_VEL
LIN {X 0,Y 601.339,Z 567.126,A -85,B 0,C 180,E1 -706.482,E2 -706.482} C_VEL
LIN {X 0,Y 601.373,Z 563.127,A -85,B 0,C 180,E1 -707.514,E2 -707.514} C_VEL
LIN {X 0,Y 601.362,Z 558.214,A -85,B 0,C 180,E1 -708.54,E2 -708.54} C_VEL
LIN {X 0,Y 601.395,Z 551.146,A -85,B 0,C 180,E1 -709.734,E2 -709.734} C_VEL
LIN {X 0,Y 601.427,Z 542.43,A -85,B 0,C 180,E1 -710.923,E2 -710.923} C_VEL
LIN {X 0,Y 601.46,Z 533.371,A -85,B 0,C 180,E1 -711.939,E2 -711.939} C_VEL
LIN {X 0,Y 601.472,Z 522.469,A -85,B 0,C 180,E1 -712.953,E2 -712.953} C_VEL
LIN {X 0,Y 601.527,Z 510.477,A -85,B 0,C 180,E1 -713.858,E2 -713.858} C_VEL
LIN {X 0,Y 601.565,Z 497.765,A -85,B 0,C 180,E1 -714.637,E2 -714.637} C_VEL
LIN {X 0,Y 601.589,Z 485.847,A -85,B 0,C 180,E1 -715.225,E2 -715.225} C_VEL
LIN {X 0,Y 601.69,Z 472.766,A -85,B 0,C 180,E1 -715.729,E2 -715.729} C_VEL
LIN {X 0,Y 601.726,Z 458.675,A -85,B 0,C 180,E1 -716.128,E2 -716.128} C_VEL
LIN {X 0,Y 601.511,Z 447.782,A -85,B 0,C 180,E1 -716.347,E2 -716.347} C_VEL
LIN {X 0,Y 601.346,Z 446.364,A -85,B 0,C 180,E1 -716.398,E2 -716.398} C_VEL
LIN {X 0,Y 601.351,Z 442.661,A -85,B 0,C 180,E1 -719.33,E2 -719.33} C_VEL
LIN {X 0,Y 601.329,Z 439.329,A -85,B 0,C 180,E1 -722.009,E2 -722.009} C_VEL
LIN {X 0,Y 601.357,Z 436.046,A -85,B 0,C 180,E1 -724.692,E2 -724.692} C_VEL
LIN {X 0,Y 601.355,Z 432.816,A -85,B 0,C 180,E1 -727.386,E2 -727.386} C_VEL
LIN {X 0,Y 601.326,Z 429.638,A -85,B 0,C 180,E1 -730.097,E2 -730.097} C_VEL
LIN {X 0,Y 601.341,Z 427.289,A -85,B 0,C 180,E1 -732.144,E2 -732.144} C_VEL
LIN {X 0,Y 601.372,Z 424.498,A -85,B 0,C 180,E1 -734.898,E2 -734.898} C_VEL
LIN {X 0,Y 601.398,Z 421.695,A -85,B 0,C 180,E1 -737.688,E2 -737.688} C_VEL
LIN {X 0,Y 601.396,Z 419.482,A -85,B 0,C 180,E1 -739.81,E2 -739.81} C_VEL
LIN {X 0,Y 601.407,Z 419.191,A -85,B 0,C 180,E1 -741.239,E2 -741.239} C_VEL
LIN {X 0,Y 601.46,Z 419.194,A -85,B 0,C 180,E1 -744.14,E2 -744.14} C_VEL
LIN {X 0,Y 601.446,Z 419.186,A -85,B 0,C 180,E1 -747.111,E2 -747.111} C_VEL
LIN {X 0,Y 601.419,Z 419.19,A -85,B 0,C 180,E1 -749.393,E2 -749.393} C_VEL
LIN {X 0,Y 601.413,Z 419.194,A -85,B 0,C 180,E1 -751.726,E2 -751.726} C_VEL
LIN {X 0,Y 601.428,Z 419.197,A -85,B 0,C 180,E1 -754.118,E2 -754.118} C_VEL
LIN {X 0,Y 601.408,Z 419.192,A -85,B 0,C 180,E1 -756.583,E2 -756.583} C_VEL
LIN {X 0,Y 601.437,Z 419.19,A -85,B 0,C 180,E1 -759.537,E2 -759.537} C_VEL
LIN {X 0,Y 601.413,Z 419.191,A -85,B 0,C 180,E1 -762.592,E2 -762.592} C_VEL
LIN {X 0,Y 601.42,Z 419.191,A -85,B 0,C 180,E1 -764.536,E2 -764.536} C_VEL
LIN {X 0,Y 601.41,Z 419.194,A -85,B 0,C 180,E1 -767.331,E2 -767.331} C_VEL
LIN {X 0,Y 601.412,Z 419.199,A -85,B 0,C 180,E1 -770.006,E2 -770.006} C_VEL
LIN {X 0,Y 601.434,Z 419.341,A -85,B 0,C 180,E1 -771.051,E2 -771.051} C_VEL
LIN {X 0,Y 601.619,Z 423.577,A -85,B 0,C 180,E1 -772.595,E2 -772.595} C_VEL
LIN {X 0,Y 601.537,Z 432.338,A -85,B 0,C 180,E1 -775.484,E2 -775.484} C_VEL
LIN {X 0,Y 601.57,Z 441.468,A -85,B 0,C 180,E1 -778.284,E2 -778.284} C_VEL
LIN {X 0,Y 601.502,Z 451.113,A -85,B 0,C 180,E1 -781.2,E2 -781.2} C_VEL
LIN {X 0,Y 601.472,Z 461.04,A -85,B 0,C 180,E1 -784.121,E2 -784.121} C_VEL
LIN {X 0,Y 601.439,Z 469.627,A -85,B 0,C 180,E1 -786.591,E2 -786.591} C_VEL
LIN {X 0,Y 601.435,Z 478.873,A -85,B 0,C 180,E1 -789.201,E2 -789.201} C_VEL
LIN {X 0,Y 601.404,Z 488.826,A -85,B 0,C 180,E1 -791.96,E2 -791.96} C_VEL
LIN {X 0,Y 601.389,Z 499.066,A -85,B 0,C 180,E1 -794.756,E2 -794.756} C_VEL
LIN {X 0,Y 601.398,Z 502.464,A -85,B 0,C 180,E1 -795.62,E2 -795.62} C_VEL
LIN {X 0,Y 601.745,Z 506.559,A -85,B 0,C 180,E1 -795.686,E2 -795.686} C_VEL
LIN {X 0,Y 601.706,Z 521.035,A -85,B 0,C 180,E1 -795.972,E2 -795.972} C_VEL
LIN {X 0,Y 601.639,Z 534.951,A -85,B 0,C 180,E1 -796.387,E2 -796.387} C_VEL
LIN {X 0,Y 601.625,Z 548.098,A -85,B 0,C 180,E1 -796.919,E2 -796.919} C_VEL
LIN {X 0,Y 601.567,Z 561.269,A -85,B 0,C 180,E1 -797.604,E2 -797.604} C_VEL
LIN {X 0,Y 601.511,Z 573.152,A -85,B 0,C 180,E1 -798.373,E2 -798.373} C_VEL
LIN {X 0,Y 601.489,Z 583.995,A -85,B 0,C 180,E1 -799.225,E2 -799.225} C_VEL
LIN {X 0,Y 601.422,Z 594.709,A -85,B 0,C 180,E1 -800.245,E2 -800.245} C_VEL
LIN {X 0,Y 601.407,Z 603.559,A -85,B 0,C 180,E1 -801.262,E2 -801.262} C_VEL
LIN {X 0,Y 601.406,Z 612.04,A -85,B 0,C 180,E1 -802.446,E2 -802.446} C_VEL
LIN {X 0,Y 601.361,Z 618.751,A -85,B 0,C 180,E1 -803.604,E2 -803.604} C_VEL
LIN {X 0,Y 601.355,Z 623.568,A -85,B 0,C 180,E1 -804.635,E2 -804.635} C_VEL
LIN {X 0,Y 601.343,Z 628.442,A -85,B 0,C 180,E1 -805.979,E2 -805.979} C_VEL
LIN {X 0,Y 601.324,Z 631.831,A -85,B 0,C 180,E1 -807.32,E2 -807.32} C_VEL
LIN {X 0,Y 601.342,Z 633.831,A -85,B 0,C 180,E1 -808.661,E2 -808.661} C_VEL
LIN {X 0,Y 601.333,Z 634.5,A -85,B 0,C 180,E1 -810,E2 -810} C_VEL
LIN {X 0,Y 601.342,Z 633.831,A -85,B 0,C 180,E1 -811.339,E2 -811.339} C_VEL
LIN {X 0,Y 601.324,Z 631.832,A -85,B 0,C 180,E1 -812.68,E2 -812.68} C_VEL
LIN {X 0,Y 601.343,Z 628.442,A -85,B 0,C 180,E1 -814.021,E2 -814.021} C_VEL
LIN {X 0,Y 601.355,Z 623.568,A -85,B 0,C 180,E1 -815.365,E2 -815.365} C_VEL
LIN {X 0,Y 601.355,Z 617.052,A -85,B 0,C 180,E1 -816.711,E2 -816.711} C_VEL
LIN {X 0,Y 601.398,Z 609.799,A -85,B 0,C 180,E1 -817.892,E2 -817.892} C_VEL
LIN {X 0,Y 601.43,Z 600.824,A -85,B 0,C 180,E1 -819.076,E2 -819.076} C_VEL
LIN {X 0,Y 601.44,Z 591.393,A -85,B 0,C 180,E1 -820.095,E2 -820.095} C_VEL
LIN {X 0,Y 601.505,Z 580.694,A -85,B 0,C 180,E1 -821.05,E2 -821.05} C_VEL
LIN {X 0,Y 601.545,Z 569.429,A -85,B 0,C 180,E1 -821.883,E2 -821.883} C_VEL
LIN {X 0,Y 601.551,Z 556.647,A -85,B 0,C 180,E1 -822.654,E2 -822.654} C_VEL
LIN {X 0,Y 601.622,Z 544.163,A -85,B 0,C 180,E1 -823.253,E2 -823.253} C_VEL
LIN {X 0,Y 601.681,Z 530.84,A -85,B 0,C 180,E1 -823.749,E2 -823.749} C_VEL
LIN {X 0,Y 601.699,Z 516.521,A -85,B 0,C 180,E1 -824.135,E2 -824.135} C_VEL
LIN {X 0,Y 601.586,Z 503.539,A -85,B 0,C 180,E1 -824.361,E2 -824.361} C_VEL
LIN {X 0,Y 601.376,Z 502.242,A -85,B 0,C 180,E1 -824.385,E2 -824.385} C_VEL
LIN {X 0,Y 601.387,Z 492.666,A -85,B 0,C 180,E1 -826.987,E2 -826.987} C_VEL
LIN {X 0,Y 601.413,Z 482.426,A -85,B 0,C 180,E1 -829.809,E2 -829.809} C_VEL
LIN {X 0,Y 601.435,Z 472.187,A -85,B 0,C 180,E1 -832.682,E2 -832.682} C_VEL
LIN {X 0,Y 601.452,Z 463.227,A -85,B 0,C 180,E1 -835.245,E2 -835.245} C_VEL
LIN {X 0,Y 601.508,Z 454.267,A -85,B 0,C 180,E1 -837.862,E2 -837.862} C_VEL
LIN {X 0,Y 601.545,Z 444.028,A -85,B 0,C 180,E1 -840.934,E2 -840.934} C_VEL
LIN {X 0,Y 601.569,Z 434.19,A -85,B 0,C 180,E1 -843.955,E2 -843.955} C_VEL
LIN {X 0,Y 601.619,Z 426.087,A -85,B 0,C 180,E1 -846.567,E2 -846.567} C_VEL
LIN {X 0,Y 601.595,Z 420.354,A -85,B 0,C 180,E1 -848.49,E2 -848.49} C_VEL
LIN {X 0,Y 601.437,Z 419.195,A -85,B 0,C 180,E1 -848.949,E2 -848.949} C_VEL
LIN {X 0,Y 601.424,Z 419.194,A -85,B 0,C 180,E1 -851.764,E2 -851.764} C_VEL
LIN {X 0,Y 601.42,Z 419.195,A -85,B 0,C 180,E1 -854.535,E2 -854.535} C_VEL
LIN {X 0,Y 601.411,Z 419.196,A -85,B 0,C 180,E1 -857.33,E2 -857.33} C_VEL
LIN {X 0,Y 601.406,Z 419.196,A -85,B 0,C 180,E1 -860.005,E2 -860.005} C_VEL
LIN {X 0,Y 601.434,Z 419.192,A -85,B 0,C 180,E1 -862.617,E2 -862.617} C_VEL
LIN {X 0,Y 601.404,Z 419.197,A -85,B 0,C 180,E1 -865.067,E2 -865.067} C_VEL
LIN {X 0,Y 601.436,Z 419.196,A -85,B 0,C 180,E1 -867.485,E2 -867.485} C_VEL
LIN {X 0,Y 601.443,Z 419.193,A -85,B 0,C 180,E1 -869.847,E2 -869.847} C_VEL
LIN {X 0,Y 601.454,Z 419.195,A -85,B 0,C 180,E1 -872.889,E2 -872.889} C_VEL
LIN {X 0,Y 601.451,Z 419.192,A -85,B 0,C 180,E1 -875.859,E2 -875.859} C_VEL
LIN {X 0,Y 601.407,Z 419.197,A -85,B 0,C 180,E1 -878.761,E2 -878.761} C_VEL
LIN {X 0,Y 601.417,Z 419.195,A -85,B 0,C 180,E1 -881.608,E2 -881.608} C_VEL
LIN {X 0,Y 601.418,Z 419.195,A -85,B 0,C 180,E1 -884.409,E2 -884.409} C_VEL
LIN {X 0,Y 601.418,Z 419.195,A -85,B 0,C 180,E1 -887.172,E2 -887.172} C_VEL
LIN {X 0,Y 601.43,Z 419.193,A -85,B 0,C 180,E1 -889.905,E2 -889.905} C_VEL
LIN {X 0,Y 601.448,Z 419.191,A -85,B 0,C 180,E1 -892.615,E2 -892.615} C_VEL
LIN {X 0,Y 601.428,Z 419.194,A -85,B 0,C 180,E1 -895.308,E2 -895.308} C_VEL
LIN {X 0,Y 601.421,Z 419.195,A -85,B 0,C 180,E1 -897.991,E2 -897.991} C_VEL
LIN {X 0,Y 601.448,Z 419.192,A -85,B 0,C 180,E1 -900.67,E2 -900.67} C_VEL
LIN {X 0,Y 601.435,Z 419.194,A -85,B 0,C 180,E1 -903.35,E2 -903.35} C_VEL
LIN {X 0,Y 601.441,Z 419.194,A -85,B 0,C 180,E1 -906.037,E2 -906.037} C_VEL
LIN {X 0,Y 601.438,Z 419.195,A -85,B 0,C 180,E1 -908.738,E2 -908.738} C_VEL
LIN {X 0,Y 601.43,Z 419.197,A -85,B 0,C 180,E1 -911.458,E2 -911.458} C_VEL
LIN {X 0,Y 601.407,Z 419.196,A -85,B 0,C 180,E1 -912.387,E2 -912.387} C_VEL
LIN {X 0,Y 600.747,Z 419.281,A -85,B 0,C 180,E1 -912.947,E2 -912.947} C_VEL
LIN {X 0,Y 597.897,Z 419.635,A -85,B 0,C 180,E1 -913.854,E2 -913.854} C_VEL
LIN {X 0,Y 595.483,Z 419.935,A -85,B 0,C 180,E1 -914.585,E2 -914.585} C_VEL
LIN {X 0,Y 594.445,Z 420.065,A -85,B 0,C 180,E1 -915.148,E2 -915.148} C_VEL
LIN {X 0,Y 594.359,Z 420.074,A -85,B 0,C 180,E1 -915.339,E2 -915.339} C_VEL
LIN {X 0,Y 594.375,Z 420.073,A -85,B 0,C 180,E1 -917.905,E2 -917.905} C_VEL
LIN {X 0,Y 594.382,Z 420.076,A -85,B 0,C 180,E1 -920.92,E2 -920.92} C_VEL
LIN {X 0,Y 594.391,Z 420.074,A -85,B 0,C 180,E1 -923.704,E2 -923.704} C_VEL
LIN {X 0,Y 594.382,Z 420.073,A -85,B 0,C 180,E1 -926.7,E2 -926.7} C_VEL
LIN {X 0,Y 594.378,Z 420.074,A -85,B 0,C 180,E1 -928.999,E2 -928.999} C_VEL
LIN {X 0,Y 594.39,Z 420.071,A -85,B 0,C 180,E1 -931.646,E2 -931.646} C_VEL
LIN {X 0,Y 594.38,Z 420.075,A -85,B 0,C 180,E1 -934.58,E2 -934.58} C_VEL
LIN {X 0,Y 594.383,Z 420.072,A -85,B 0,C 180,E1 -937.087,E2 -937.087} C_VEL
LIN {X 0,Y 594.356,Z 420.075,A -85,B 0,C 180,E1 -939.773,E2 -939.773} C_VEL
LIN {X 0,Y 594.387,Z 420.07,A -85,B 0,C 180,E1 -942.374,E2 -942.374} C_VEL
LIN {X 0,Y 594.361,Z 420.073,A -85,B 0,C 180,E1 -945.192,E2 -945.192} C_VEL
LIN {X 0,Y 594.366,Z 420.073,A -85,B 0,C 180,E1 -947.625,E2 -947.625} C_VEL
LIN {X 0,Y 594.393,Z 420.07,A -85,B 0,C 180,E1 -950.322,E2 -950.322} C_VEL
LIN {X 0,Y 594.385,Z 420.072,A -85,B 0,C 180,E1 -952.914,E2 -952.914} C_VEL
LIN {X 0,Y 594.388,Z 420.07,A -85,B 0,C 180,E1 -955.861,E2 -955.861} C_VEL
LIN {X 0,Y 594.371,Z 420.072,A -85,B 0,C 180,E1 -958.65,E2 -958.65} C_VEL
LIN {X 0,Y 594.385,Z 420.073,A -85,B 0,C 180,E1 -961.043,E2 -961.043} C_VEL
LIN {X 0,Y 594.391,Z 420.07,A -85,B 0,C 180,E1 -963.977,E2 -963.977} C_VEL
LIN {X 0,Y 594.39,Z 420.075,A -85,B 0,C 180,E1 -966.296,E2 -966.296} C_VEL
LIN {X 0,Y 594.403,Z 420.071,A -85,B 0,C 180,E1 -969.225,E2 -969.225} C_VEL
LIN {X 0,Y 594.357,Z 420.076,A -85,B 0,C 180,E1 -972.095,E2 -972.095} C_VEL
LIN {X 0,Y 594.369,Z 420.074,A -85,B 0,C 180,E1 -974.219,E2 -974.219} C_VEL
LIN {X 0,Y 594.384,Z 420.071,A -85,B 0,C 180,E1 -976.321,E2 -976.321} C_VEL
LIN {X 0,Y 594.376,Z 420.072,A -85,B 0,C 180,E1 -979.095,E2 -979.095} C_VEL
LIN {X 0,Y 594.418,Z 420.067,A -85,B 0,C 180,E1 -981.844,E2 -981.844} C_VEL
LIN {X 0,Y 594.394,Z 420.07,A -85,B 0,C 180,E1 -984.572,E2 -984.572} C_VEL
LIN {X 0,Y 594.404,Z 420.069,A -85,B 0,C 180,E1 -987.289,E2 -987.289} C_VEL
LIN {X 0,Y 594.419,Z 420.067,A -85,B 0,C 180,E1 -990,E2 -990} C_VEL
LIN {X 0,Y 594.408,Z 420.069,A -85,B 0,C 180,E1 -992.711,E2 -992.711} C_VEL
LIN {X 0,Y 594.4,Z 420.071,A -85,B 0,C 180,E1 -995.428,E2 -995.428} C_VEL
LIN {X 0,Y 594.396,Z 420.07,A -85,B 0,C 180,E1 -997.473,E2 -997.473} C_VEL
LIN {X 0,Y 594.399,Z 420.069,A -85,B 0,C 180,E1 -1000.216,E2 -1000.216} C_VEL
LIN {X 0,Y 594.365,Z 420.074,A -85,B 0,C 180,E1 -1002.983,E2 -1002.983} C_VEL
LIN {X 0,Y 594.374,Z 420.074,A -85,B 0,C 180,E1 -1005.078,E2 -1005.078} C_VEL
LIN {X 0,Y 594.381,Z 420.072,A -85,B 0,C 180,E1 -1007.193,E2 -1007.193} C_VEL
LIN {X 0,Y 594.375,Z 420.074,A -85,B 0,C 180,E1 -1010.053,E2 -1010.053} C_VEL
LIN {X 0,Y 594.368,Z 420.077,A -85,B 0,C 180,E1 -1012.967,E2 -1012.967} C_VEL
LIN {X 0,Y 594.379,Z 420.071,A -85,B 0,C 180,E1 -1015.192,E2 -1015.192} C_VEL
LIN {X 0,Y 594.388,Z 420.071,A -85,B 0,C 180,E1 -1017.526,E2 -1017.526} C_VEL
LIN {X 0,Y 594.389,Z 420.071,A -85,B 0,C 180,E1 -1020.328,E2 -1020.328} C_VEL
LIN {X 0,Y 594.379,Z 420.073,A -85,B 0,C 180,E1 -1022.949,E2 -1022.949} C_VEL
LIN {X 0,Y 594.308,Z 420.085,A -85,B 0,C 180,E1 -1024.584,E2 -1024.584} C_VEL
LIN {X 0,Y 594.293,Z 422.654,A -85,B 0,C 180,E1 -1027.093,E2 -1027.093} C_VEL
LIN {X 0,Y 594.279,Z 425.472,A -85,B 0,C 180,E1 -1029.763,E2 -1029.763} C_VEL
LIN {X 0,Y 594.285,Z 428.743,A -85,B 0,C 180,E1 -1032.843,E2 -1032.843} C_VEL
LIN {X 0,Y 594.277,Z 432.085,A -85,B 0,C 180,E1 -1035.753,E2 -1035.753} C_VEL
LIN {X 0,Y 594.248,Z 434.919,A -85,B 0,C 180,E1 -1038.165,E2 -1038.165} C_VEL
LIN {X 0,Y 594.231,Z 437.483,A -85,B 0,C 180,E1 -1040.308,E2 -1040.308} C_VEL
LIN {X 0,Y 594.216,Z 440.635,A -85,B 0,C 180,E1 -1042.901,E2 -1042.901} C_VEL
LIN {X 0,Y 594.239,Z 444.317,A -85,B 0,C 180,E1 -1045.88,E2 -1045.88} C_VEL
LIN {X 0,Y 594.247,Z 446.416,A -85,B 0,C 180,E1 -1047.545,E2 -1047.545} C_VEL
LIN {X 0,Y 594.862,Z 451.302,A -85,B 0,C 180,E1 -1047.641,E2 -1047.641} C_VEL
LIN {X 0,Y 594.784,Z 465.59,A -85,B 0,C 180,E1 -1047.974,E2 -1047.974} C_VEL
LIN {X 0,Y 594.71,Z 479.09,A -85,B 0,C 180,E1 -1048.427,E2 -1048.427} C_VEL
LIN {X 0,Y 594.671,Z 491.275,A -85,B 0,C 180,E1 -1048.964,E2 -1048.964} C_VEL
LIN {X 0,Y 594.585,Z 503.498,A -85,B 0,C 180,E1 -1049.638,E2 -1049.638} C_VEL
LIN {X 0,Y 594.515,Z 515.128,A -85,B 0,C 180,E1 -1050.426,E2 -1050.426} C_VEL
LIN {X 0,Y 594.455,Z 526.812,A -85,B 0,C 180,E1 -1051.392,E2 -1051.392} C_VEL
LIN {X 0,Y 594.369,Z 536.54,A -85,B 0,C 180,E1 -1052.367,E2 -1052.367} C_VEL
LIN {X 0,Y 594.342,Z 545.754,A -85,B 0,C 180,E1 -1053.487,E2 -1053.487} C_VEL
LIN {X 0,Y 594.311,Z 553.384,A -85,B 0,C 180,E1 -1054.616,E2 -1054.616} C_VEL
LIN {X 0,Y 594.278,Z 558.829,A -85,B 0,C 180,E1 -1055.588,E2 -1055.588} C_VEL
LIN {X 0,Y 594.271,Z 563.752,A -85,B 0,C 180,E1 -1056.66,E2 -1056.66} C_VEL
LIN {X 0,Y 594.263,Z 567.777,A -85,B 0,C 180,E1 -1057.762,E2 -1057.762} C_VEL
LIN {X 0,Y 594.25,Z 571.589,A -85,B 0,C 180,E1 -1059.219,E2 -1059.219} C_VEL
LIN {X 0,Y 594.209,Z 573.797,A -85,B 0,C 180,E1 -1060.66,E2 -1060.66} C_VEL
LIN {X 0,Y 594.249,Z 574.338,A -85,B 0,C 180,E1 -1061.378,E2 -1061.378} C_VEL
LIN {X 0,Y 594.235,Z 574.278,A -85,B 0,C 180,E1 -1062.802,E2 -1062.802} C_VEL
LIN {X 0,Y 594.249,Z 572.777,A -85,B 0,C 180,E1 -1064.216,E2 -1064.216} C_VEL
LIN {X 0,Y 594.243,Z 569.835,A -85,B 0,C 180,E1 -1065.619,E2 -1065.619} C_VEL
LIN {X 0,Y 594.257,Z 565.396,A -85,B 0,C 180,E1 -1067.014,E2 -1067.014} C_VEL
LIN {X 0,Y 594.264,Z 560.999,A -85,B 0,C 180,E1 -1068.055,E2 -1068.055} C_VEL
LIN {X 0,Y 594.286,Z 554.619,A -85,B 0,C 180,E1 -1069.265,E2 -1069.265} C_VEL
LIN {X 0,Y 594.32,Z 546.711,A -85,B 0,C 180,E1 -1070.47,E2 -1070.47} C_VEL
LIN {X 0,Y 594.357,Z 538.49,A -85,B 0,C 180,E1 -1071.5,E2 -1071.5} C_VEL
LIN {X 0,Y 594.452,Z 528.631,A -85,B 0,C 180,E1 -1072.527,E2 -1072.527} C_VEL
LIN {X 0,Y 594.506,Z 517.61,A -85,B 0,C 180,E1 -1073.478,E2 -1073.478} C_VEL
LIN {X 0,Y 594.559,Z 505.689,A -85,B 0,C 180,E1 -1074.318,E2 -1074.318} C_VEL
LIN {X 0,Y 594.654,Z 493.83,A -85,B 0,C 180,E1 -1074.999,E2 -1074.999} C_VEL
LIN {X 0,Y 594.716,Z 480.847,A -85,B 0,C 180,E1 -1075.594,E2 -1075.594} C_VEL
LIN {X 0,Y 594.792,Z 466.728,A -85,B 0,C 180,E1 -1076.083,E2 -1076.083} C_VEL
LIN {X 0,Y 594.854,Z 452.684,A -85,B 0,C 180,E1 -1076.422,E2 -1076.422} C_VEL
LIN {X 0,Y 594.607,Z 448.519,A -85,B 0,C 180,E1 -1076.506,E2 -1076.506} C_VEL
LIN {X 0,Y 594.251,Z 446.398,A -85,B 0,C 180,E1 -1076.546,E2 -1076.546} C_VEL
LIN {X 0,Y 594.256,Z 442.934,A -85,B 0,C 180,E1 -1079.322,E2 -1079.322} C_VEL
LIN {X 0,Y 594.235,Z 439.603,A -85,B 0,C 180,E1 -1082.033,E2 -1082.033} C_VEL
LIN {X 0,Y 594.277,Z 436.32,A -85,B 0,C 180,E1 -1084.748,E2 -1084.748} C_VEL
LIN {X 0,Y 594.27,Z 433.091,A -85,B 0,C 180,E1 -1087.475,E2 -1087.475} C_VEL
LIN {X 0,Y 594.238,Z 429.916,A -85,B 0,C 180,E1 -1090.218,E2 -1090.218} C_VEL
LIN {X 0,Y 594.265,Z 427.63,A -85,B 0,C 180,E1 -1092.291,E2 -1092.291} C_VEL
LIN {X 0,Y 594.287,Z 425.703,A -85,B 0,C 180,E1 -1094.379,E2 -1094.379} C_VEL
LIN {X 0,Y 594.308,Z 422.882,A -85,B 0,C 180,E1 -1097.196,E2 -1097.196} C_VEL
LIN {X 0,Y 594.321,Z 420.673,A -85,B 0,C 180,E1 -1099.336,E2 -1099.336} C_VEL
LIN {X 0,Y 594.328,Z 420.083,A -85,B 0,C 180,E1 -1100.055,E2 -1100.055} C_VEL
LIN {X 0,Y 594.36,Z 420.071,A -85,B 0,C 180,E1 -1102.736,E2 -1102.736} C_VEL
LIN {X 0,Y 594.373,Z 420.067,A -85,B 0,C 180,E1 -1105.193,E2 -1105.193} C_VEL
LIN {X 0,Y 594.379,Z 420.068,A -85,B 0,C 180,E1 -1107.527,E2 -1107.527} C_VEL
LIN {X 0,Y 594.395,Z 420.07,A -85,B 0,C 180,E1 -1110.331,E2 -1110.331} C_VEL
LIN {X 0,Y 594.375,Z 420.067,A -85,B 0,C 180,E1 -1112.95,E2 -1112.95} C_VEL
LIN {X 0,Y 594.377,Z 420.068,A -85,B 0,C 180,E1 -1115.407,E2 -1115.407} C_VEL
LIN {X 0,Y 594.385,Z 420.075,A -85,B 0,C 180,E1 -1117.941,E2 -1117.941} C_VEL
LIN {X 0,Y 594.376,Z 420.067,A -85,B 0,C 180,E1 -1120.823,E2 -1120.823} C_VEL
LIN {X 0,Y 594.38,Z 420.076,A -85,B 0,C 180,E1 -1123.842,E2 -1123.842} C_VEL
LIN {X 0,Y 594.376,Z 420.068,A -85,B 0,C 180,E1 -1126.702,E2 -1126.702} C_VEL
LIN {X 0,Y 594.371,Z 420.074,A -85,B 0,C 180,E1 -1129.434,E2 -1129.434} C_VEL
LIN {X 0,Y 594.413,Z 420.159,A -85,B 0,C 180,E1 -1130.762,E2 -1130.762} C_VEL
LIN {X 0,Y 594.671,Z 424.408,A -85,B 0,C 180,E1 -1132.356,E2 -1132.356} C_VEL
LIN {X 0,Y 594.595,Z 432.305,A -85,B 0,C 180,E1 -1135.039,E2 -1135.039} C_VEL
LIN {X 0,Y 594.565,Z 441.36,A -85,B 0,C 180,E1 -1137.866,E2 -1137.866} C_VEL
LIN {X 0,Y 594.537,Z 449.148,A -85,B 0,C 180,E1 -1140.233,E2 -1140.233} C_VEL
LIN {X 0,Y 594.468,Z 458.107,A -85,B 0,C 180,E1 -1142.925,E2 -1142.925} C_VEL
LIN {X 0,Y 594.436,Z 467.067,A -85,B 0,C 180,E1 -1145.556,E2 -1145.556} C_VEL
LIN {X 0,Y 594.407,Z 476.027,A -85,B 0,C 180,E1 -1148.134,E2 -1148.134} C_VEL
LIN {X 0,Y 594.357,Z 486.46,A -85,B 0,C 180,E1 -1151.079,E2 -1151.079} C_VEL
LIN {X 0,Y 594.316,Z 496.506,A -85,B 0,C 180,E1 -1153.866,E2 -1153.866} C_VEL
LIN {X 0,Y 594.324,Z 502.244,A -85,B 0,C 180,E1 -1155.441,E2 -1155.441} C_VEL
LIN {X 0,Y 594.877,Z 506.899,A -85,B 0,C 180,E1 -1155.522,E2 -1155.522} C_VEL
LIN {X 0,Y 594.814,Z 521.346,A -85,B 0,C 180,E1 -1155.814,E2 -1155.814} C_VEL
LIN {X 0,Y 594.757,Z 534.136,A -85,B 0,C 180,E1 -1156.199,E2 -1156.199} C_VEL
LIN {X 0,Y 594.686,Z 548.099,A -85,B 0,C 180,E1 -1156.764,E2 -1156.764} C_VEL
LIN {X 0,Y 594.604,Z 561.268,A -85,B 0,C 180,E1 -1157.456,E2 -1157.456} C_VEL
LIN {X 0,Y 594.534,Z 573.152,A -85,B 0,C 180,E1 -1158.234,E2 -1158.234} C_VEL
LIN {X 0,Y 594.475,Z 583.995,A -85,B 0,C 180,E1 -1159.097,E2 -1159.097} C_VEL
LIN {X 0,Y 594.375,Z 594.709,A -85,B 0,C 180,E1 -1160.128,E2 -1160.128} C_VEL
LIN {X 0,Y 594.351,Z 603.559,A -85,B 0,C 180,E1 -1161.158,E2 -1161.158} C_VEL
LIN {X 0,Y 594.316,Z 612.04,A -85,B 0,C 180,E1 -1162.355,E2 -1162.355} C_VEL
LIN {X 0,Y 594.27,Z 619.233,A -85,B 0,C 180,E1 -1163.619,E2 -1163.619} C_VEL
LIN {X 0,Y 594.248,Z 624.962,A -85,B 0,C 180,E1 -1164.911,E2 -1164.911} C_VEL
LIN {X 0,Y 594.259,Z 628.442,A -85,B 0,C 180,E1 -1165.931,E2 -1165.931} C_VEL
LIN {X 0,Y 594.224,Z 631.831,A -85,B 0,C 180,E1 -1167.288,E2 -1167.288} C_VEL
LIN {X 0,Y 594.242,Z 633.831,A -85,B 0,C 180,E1 -1168.645,E2 -1168.645} C_VEL
LIN {X 0,Y 594.234,Z 634.5,A -85,B 0,C 180,E1 -1170,E2 -1170} C_VEL
LIN {X 0,Y 594.242,Z 633.831,A -85,B 0,C 180,E1 -1171.355,E2 -1171.355} C_VEL
LIN {X 0,Y 594.224,Z 631.832,A -85,B 0,C 180,E1 -1172.712,E2 -1172.712} C_VEL
LIN {X 0,Y 594.259,Z 628.443,A -85,B 0,C 180,E1 -1174.069,E2 -1174.069} C_VEL
LIN {X 0,Y 594.275,Z 623.568,A -85,B 0,C 180,E1 -1175.429,E2 -1175.429} C_VEL
LIN {X 0,Y 594.299,Z 618.033,A -85,B 0,C 180,E1 -1176.607,E2 -1176.607} C_VEL
LIN {X 0,Y 594.316,Z 610.92,A -85,B 0,C 180,E1 -1177.816,E2 -1177.816} C_VEL
LIN {X 0,Y 594.369,Z 602.2,A -85,B 0,C 180,E1 -1179.014,E2 -1179.014} C_VEL
LIN {X 0,Y 594.4,Z 593.083,A -85,B 0,C 180,E1 -1180.044,E2 -1180.044} C_VEL
LIN {X 0,Y 594.478,Z 582.703,A -85,B 0,C 180,E1 -1181.017,E2 -1181.017} C_VEL
LIN {X 0,Y 594.575,Z 570.708,A -85,B 0,C 180,E1 -1181.938,E2 -1181.938} C_VEL
LIN {X 0,Y 594.605,Z 558.215,A -85,B 0,C 180,E1 -1182.717,E2 -1182.717} C_VEL
LIN {X 0,Y 594.686,Z 546.134,A -85,B 0,C 180,E1 -1183.323,E2 -1183.323} C_VEL
LIN {X 0,Y 594.779,Z 532.184,A -85,B 0,C 180,E1 -1183.866,E2 -1183.866} C_VEL
LIN {X 0,Y 594.841,Z 518.278,A -85,B 0,C 180,E1 -1184.259,E2 -1184.259} C_VEL
LIN {X 0,Y 594.737,Z 504.571,A -85,B 0,C 180,E1 -1184.515,E2 -1184.515} C_VEL
LIN {X 0,Y 594.341,Z 502.232,A -85,B 0,C 180,E1 -1184.562,E2 -1184.562} C_VEL
LIN {X 0,Y 594.336,Z 491.386,A -85,B 0,C 180,E1 -1187.55,E2 -1187.55} C_VEL
LIN {X 0,Y 594.38,Z 481.146,A -85,B 0,C 180,E1 -1190.414,E2 -1190.414} C_VEL
LIN {X 0,Y 594.416,Z 472.187,A -85,B 0,C 180,E1 -1192.965,E2 -1192.965} C_VEL
LIN {X 0,Y 594.466,Z 463.227,A -85,B 0,C 180,E1 -1195.563,E2 -1195.563} C_VEL
LIN {X 0,Y 594.499,Z 454.267,A -85,B 0,C 180,E1 -1198.22,E2 -1198.22} C_VEL
LIN {X 0,Y 594.569,Z 445.308,A -85,B 0,C 180,E1 -1200.942,E2 -1200.942} C_VEL
LIN {X 0,Y 594.567,Z 436.211,A -85,B 0,C 180,E1 -1203.748,E2 -1203.748} C_VEL
LIN {X 0,Y 594.654,Z 428.607,A -85,B 0,C 180,E1 -1206.222,E2 -1206.222} C_VEL
LIN {X 0,Y 594.704,Z 422.403,A -85,B 0,C 180,E1 -1208.316,E2 -1208.316} C_VEL
LIN {X 0,Y 594.408,Z 420.072,A -85,B 0,C 180,E1 -1209.184,E2 -1209.184} C_VEL
LIN {X 0,Y 594.382,Z 420.072,A -85,B 0,C 180,E1 -1211.848,E2 -1211.848} C_VEL
LIN {X 0,Y 594.36,Z 420.077,A -85,B 0,C 180,E1 -1214.808,E2 -1214.808} C_VEL
LIN {X 0,Y 594.369,Z 420.076,A -85,B 0,C 180,E1 -1217.625,E2 -1217.625} C_VEL
LIN {X 0,Y 594.385,Z 420.073,A -85,B 0,C 180,E1 -1220.32,E2 -1220.32} C_VEL
LIN {X 0,Y 594.384,Z 420.072,A -85,B 0,C 180,E1 -1222.913,E2 -1222.913} C_VEL
LIN {X 0,Y 594.38,Z 420.074,A -85,B 0,C 180,E1 -1225.86,E2 -1225.86} C_VEL
LIN {X 0,Y 594.386,Z 420.074,A -85,B 0,C 180,E1 -1228.651,E2 -1228.651} C_VEL
LIN {X 0,Y 594.383,Z 420.071,A -85,B 0,C 180,E1 -1231.04,E2 -1231.04} C_VEL
LIN {X 0,Y 594.393,Z 420.071,A -85,B 0,C 180,E1 -1233.974,E2 -1233.974} C_VEL
LIN {X 0,Y 594.385,Z 420.07,A -85,B 0,C 180,E1 -1236.296,E2 -1236.296} C_VEL
LIN {X 0,Y 594.401,Z 420.069,A -85,B 0,C 180,E1 -1239.224,E2 -1239.224} C_VEL
LIN {X 0,Y 594.376,Z 420.072,A -85,B 0,C 180,E1 -1242.096,E2 -1242.096} C_VEL
LIN {X 0,Y 594.371,Z 420.074,A -85,B 0,C 180,E1 -1244.219,E2 -1244.219} C_VEL
LIN {X 0,Y 594.365,Z 420.074,A -85,B 0,C 180,E1 -1247.017,E2 -1247.017} C_VEL
LIN {X 0,Y 594.391,Z 420.07,A -85,B 0,C 180,E1 -1249.784,E2 -1249.784} C_VEL
LIN {X 0,Y 594.397,Z 420.07,A -85,B 0,C 180,E1 -1252.527,E2 -1252.527} C_VEL
LIN {X 0,Y 594.397,Z 420.07,A -85,B 0,C 180,E1 -1255.253,E2 -1255.253} C_VEL
LIN {X 0,Y 594.391,Z 420.071,A -85,B 0,C 180,E1 -1257.967,E2 -1257.967} C_VEL
LIN {X 0,Y 594.419,Z 420.068,A -85,B 0,C 180,E1 -1260.678,E2 -1260.678} C_VEL
LIN {X 0,Y 594.385,Z 420.072,A -85,B 0,C 180,E1 -1263.389,E2 -1263.389} C_VEL
LIN {X 0,Y 594.394,Z 420.072,A -85,B 0,C 180,E1 -1266.109,E2 -1266.109} C_VEL
LIN {X 0,Y 594.398,Z 420.071,A -85,B 0,C 180,E1 -1268.842,E2 -1268.842} C_VEL
LIN {X 0,Y 594.388,Z 420.072,A -85,B 0,C 180,E1 -1271.596,E2 -1271.596} C_VEL
LIN {X 0,Y 594.384,Z 420.073,A -85,B 0,C 180,E1 -1274.377,E2 -1274.377} C_VEL
LIN {X 0,Y 594.359,Z 420.074,A -85,B 0,C 180,E1 -1275.339,E2 -1275.339} C_VEL
LIN {X 0,Y 593.689,Z 420.159,A -85,B 0,C 180,E1 -1275.905,E2 -1275.905} C_VEL
LIN {X 0,Y 590.834,Z 420.518,A -85,B 0,C 180,E1 -1276.823,E2 -1276.823} C_VEL
LIN {X 0,Y 588.428,Z 420.818,A -85,B 0,C 180,E1 -1277.562,E2 -1277.562} C_VEL
LIN {X 0,Y 587.401,Z 420.944,A -85,B 0,C 180,E1 -1278.132,E2 -1278.132} C_VEL
LIN {X 0,Y 587.32,Z 420.952,A -85,B 0,C 180,E1 -1278.325,E2 -1278.325} C_VEL
LIN {X 0,Y 587.352,Z 420.951,A -85,B 0,C 180,E1 -1281.045,E2 -1281.045} C_VEL
LIN {X 0,Y 587.335,Z 420.951,A -85,B 0,C 180,E1 -1284.007,E2 -1284.007} C_VEL
LIN {X 0,Y 587.335,Z 420.951,A -85,B 0,C 180,E1 -1286.279,E2 -1286.279} C_VEL
LIN {X 0,Y 587.346,Z 420.951,A -85,B 0,C 180,E1 -1289.135,E2 -1289.135} C_VEL
LIN {X 0,Y 587.354,Z 420.95,A -85,B 0,C 180,E1 -1291.839,E2 -1291.839} C_VEL
LIN {X 0,Y 587.348,Z 420.948,A -85,B 0,C 180,E1 -1294.349,E2 -1294.349} C_VEL
LIN {X 0,Y 587.349,Z 420.947,A -85,B 0,C 180,E1 -1296.747,E2 -1296.747} C_VEL
LIN {X 0,Y 587.33,Z 420.95,A -85,B 0,C 180,E1 -1299.361,E2 -1299.361} C_VEL
LIN {X 0,Y 587.335,Z 420.949,A -85,B 0,C 180,E1 -1302.109,E2 -1302.109} C_VEL
LIN {X 0,Y 587.314,Z 420.951,A -85,B 0,C 180,E1 -1305.09,E2 -1305.09} C_VEL
LIN {X 0,Y 587.322,Z 420.951,A -85,B 0,C 180,E1 -1307.926,E2 -1307.926} C_VEL
LIN {X 0,Y 587.346,Z 420.947,A -85,B 0,C 180,E1 -1310.642,E2 -1310.642} C_VEL
LIN {X 0,Y 587.354,Z 420.946,A -85,B 0,C 180,E1 -1313.292,E2 -1313.292} C_VEL
LIN {X 0,Y 587.37,Z 420.945,A -85,B 0,C 180,E1 -1315.781,E2 -1315.781} C_VEL
LIN {X 0,Y 587.341,Z 420.951,A -85,B 0,C 180,E1 -1318.232,E2 -1318.232} C_VEL
LIN {X 0,Y 587.353,Z 420.951,A -85,B 0,C 180,E1 -1320.867,E2 -1320.867} C_VEL
LIN {X 0,Y 587.363,Z 420.947,A -85,B 0,C 180,E1 -1323.819,E2 -1323.819} C_VEL
LIN {X 0,Y 587.338,Z 420.95,A -85,B 0,C 180,E1 -1325.994,E2 -1325.994} C_VEL
LIN {X 0,Y 587.325,Z 420.95,A -85,B 0,C 180,E1 -1328.226,E2 -1328.226} C_VEL
LIN {X 0,Y 587.351,Z 420.947,A -85,B 0,C 180,E1 -1331.152,E2 -1331.152} C_VEL
LIN {X 0,Y 587.327,Z 420.95,A -85,B 0,C 180,E1 -1334.025,E2 -1334.025} C_VEL
LIN {X 0,Y 587.362,Z 420.947,A -85,B 0,C 180,E1 -1336.155,E2 -1336.155} C_VEL
LIN {X 0,Y 587.343,Z 420.95,A -85,B 0,C 180,E1 -1338.963,E2 -1338.963} C_VEL
LIN {X 0,Y 587.37,Z 420.946,A -85,B 0,C 180,E1 -1341.745,E2 -1341.745} C_VEL
LIN {X 0,Y 587.36,Z 420.947,A -85,B 0,C 180,E1 -1344.507,E2 -1344.507} C_VEL
LIN {X 0,Y 587.371,Z 420.946,A -85,B 0,C 180,E1 -1347.257,E2 -1347.257} C_VEL
LIN {X 0,Y 587.388,Z 420.943,A -85,B 0,C 180,E1 -1350,E2 -1350} C_VEL
LIN {X 0,Y 587.375,Z 420.945,A -85,B 0,C 180,E1 -1352.743,E2 -1352.743} C_VEL
LIN {X 0,Y 587.365,Z 420.946,A -85,B 0,C 180,E1 -1355.493,E2 -1355.493} C_VEL
LIN {X 0,Y 587.347,Z 420.948,A -85,B 0,C 180,E1 -1358.255,E2 -1358.255} C_VEL
LIN {X 0,Y 587.353,Z 420.947,A -85,B 0,C 180,E1 -1361.133,E2 -1361.133} C_VEL
LIN {X 0,Y 587.37,Z 420.944,A -85,B 0,C 180,E1 -1364.26,E2 -1364.26} C_VEL
LIN {X 0,Y 587.347,Z 420.951,A -85,B 0,C 180,E1 -1367.406,E2 -1367.406} C_VEL
LIN {X 0,Y 587.331,Z 420.954,A -85,B 0,C 180,E1 -1370.304,E2 -1370.304} C_VEL
LIN {X 0,Y 587.326,Z 420.952,A -85,B 0,C 180,E1 -1373.258,E2 -1373.258} C_VEL
LIN {X 0,Y 587.337,Z 420.951,A -85,B 0,C 180,E1 -1375.516,E2 -1375.516} C_VEL
LIN {X 0,Y 587.352,Z 420.946,A -85,B 0,C 180,E1 -1377.817,E2 -1377.817} C_VEL
LIN {X 0,Y 587.344,Z 420.948,A -85,B 0,C 180,E1 -1380.51,E2 -1380.51} C_VEL
LIN {X 0,Y 587.337,Z 420.949,A -85,B 0,C 180,E1 -1383.111,E2 -1383.111} C_VEL
LIN {X 0,Y 587.226,Z 421.149,A -85,B 0,C 180,E1 -1385.062,E2 -1385.062} C_VEL
LIN {X 0,Y 587.214,Z 424.006,A -85,B 0,C 180,E1 -1387.822,E2 -1387.822} C_VEL
LIN {X 0,Y 587.183,Z 426.549,A -85,B 0,C 180,E1 -1390.264,E2 -1390.264} C_VEL
LIN {X 0,Y 587.203,Z 429.481,A -85,B 0,C 180,E1 -1393.106,E2 -1393.106} C_VEL
LIN {X 0,Y 587.188,Z 432.803,A -85,B 0,C 180,E1 -1396.036,E2 -1396.036} C_VEL
LIN {X 0,Y 587.155,Z 436.195,A -85,B 0,C 180,E1 -1398.944,E2 -1398.944} C_VEL
LIN {X 0,Y 587.129,Z 439.243,A -85,B 0,C 180,E1 -1401.505,E2 -1401.505} C_VEL
LIN {X 0,Y 587.129,Z 442.852,A -85,B 0,C 180,E1 -1404.484,E2 -1404.484} C_VEL
LIN {X 0,Y 587.163,Z 446.387,A -85,B 0,C 180,E1 -1407.356,E2 -1407.356} C_VEL
LIN {X 0,Y 587.981,Z 452.046,A -85,B 0,C 180,E1 -1407.483,E2 -1407.483} C_VEL
LIN {X 0,Y 587.892,Z 466.782,A -85,B 0,C 180,E1 -1407.841,E2 -1407.841} C_VEL
LIN {X 0,Y 587.789,Z 480.219,A -85,B 0,C 180,E1 -1408.308,E2 -1408.308} C_VEL
LIN {X 0,Y 587.738,Z 492.276,A -85,B 0,C 180,E1 -1408.857,E2 -1408.857} C_VEL
LIN {X 0,Y 587.617,Z 505.022,A -85,B 0,C 180,E1 -1409.583,E2 -1409.583} C_VEL
LIN {X 0,Y 587.51,Z 517.077,A -85,B 0,C 180,E1 -1410.432,E2 -1410.432} C_VEL
LIN {X 0,Y 587.432,Z 528.35,A -85,B 0,C 180,E1 -1411.409,E2 -1411.409} C_VEL
LIN {X 0,Y 587.331,Z 538.195,A -85,B 0,C 180,E1 -1412.441,E2 -1412.441} C_VEL
LIN {X 0,Y 587.276,Z 546.776,A -85,B 0,C 180,E1 -1413.527,E2 -1413.527} C_VEL
LIN {X 0,Y 587.238,Z 554.215,A -85,B 0,C 180,E1 -1414.668,E2 -1414.668} C_VEL
LIN {X 0,Y 587.221,Z 561.12,A -85,B 0,C 180,E1 -1415.988,E2 -1415.988} C_VEL
LIN {X 0,Y 587.175,Z 565.925,A -85,B 0,C 180,E1 -1417.163,E2 -1417.163} C_VEL
LIN {X 0,Y 587.167,Z 569.297,A -85,B 0,C 180,E1 -1418.219,E2 -1418.219} C_VEL
LIN {X 0,Y 587.166,Z 571.209,A -85,B 0,C 180,E1 -1419.002,E2 -1419.002} C_VEL
LIN {X 0,Y 587.113,Z 573.541,A -85,B 0,C 180,E1 -1420.417,E2 -1420.417} C_VEL
LIN {X 0,Y 587.124,Z 574.466,A -85,B 0,C 180,E1 -1421.867,E2 -1421.867} C_VEL
LIN {X 0,Y 587.156,Z 573.939,A -85,B 0,C 180,E1 -1423.305,E2 -1423.305} C_VEL
LIN {X 0,Y 587.141,Z 571.952,A -85,B 0,C 180,E1 -1424.732,E2 -1424.732} C_VEL
LIN {X 0,Y 587.178,Z 568.484,A -85,B 0,C 180,E1 -1426.15,E2 -1426.15} C_VEL
LIN {X 0,Y 587.196,Z 563.489,A -85,B 0,C 180,E1 -1427.559,E2 -1427.559} C_VEL
LIN {X 0,Y 587.222,Z 557.021,A -85,B 0,C 180,E1 -1428.925,E2 -1428.925} C_VEL
LIN {X 0,Y 587.278,Z 549.457,A -85,B 0,C 180,E1 -1430.181,E2 -1430.181} C_VEL
LIN {X 0,Y 587.299,Z 540.353,A -85,B 0,C 180,E1 -1431.397,E2 -1431.397} C_VEL
LIN {X 0,Y 587.407,Z 530.845,A -85,B 0,C 180,E1 -1432.437,E2 -1432.437} C_VEL
LIN {X 0,Y 587.487,Z 519.865,A -85,B 0,C 180,E1 -1433.431,E2 -1433.431} C_VEL
LIN {X 0,Y 587.6,Z 507.638,A -85,B 0,C 180,E1 -1434.337,E2 -1434.337} C_VEL
LIN {X 0,Y 587.71,Z 494.661,A -85,B 0,C 180,E1 -1435.112,E2 -1435.112} C_VEL
LIN {X 0,Y 587.81,Z 481.915,A -85,B 0,C 180,E1 -1435.714,E2 -1435.714} C_VEL
LIN {X 0,Y 587.903,Z 468.183,A -85,B 0,C 180,E1 -1436.209,E2 -1436.209} C_VEL
LIN {X 0,Y 587.971,Z 453.767,A -85,B 0,C 180,E1 -1436.574,E2 -1436.574} C_VEL
LIN {X 0,Y 587.648,Z 449.294,A -85,B 0,C 180,E1 -1436.668,E2 -1436.668} C_VEL
LIN {X 0,Y 587.157,Z 446.379,A -85,B 0,C 180,E1 -1436.741,E2 -1436.741} C_VEL
LIN {X 0,Y 587.16,Z 443.208,A -85,B 0,C 180,E1 -1439.314,E2 -1439.314} C_VEL
LIN {X 0,Y 587.141,Z 439.876,A -85,B 0,C 180,E1 -1442.058,E2 -1442.058} C_VEL
LIN {X 0,Y 587.183,Z 436.595,A -85,B 0,C 180,E1 -1444.806,E2 -1444.806} C_VEL
LIN {X 0,Y 587.184,Z 433.367,A -85,B 0,C 180,E1 -1447.565,E2 -1447.565} C_VEL
LIN {X 0,Y 587.153,Z 430.194,A -85,B 0,C 180,E1 -1450.343,E2 -1450.343} C_VEL
LIN {X 0,Y 587.209,Z 428.275,A -85,B 0,C 180,E1 -1452.441,E2 -1452.441} C_VEL
LIN {X 0,Y 587.253,Z 425.478,A -85,B 0,C 180,E1 -1455.265,E2 -1455.265} C_VEL
LIN {X 0,Y 587.269,Z 423.376,A -85,B 0,C 180,E1 -1457.408,E2 -1457.408} C_VEL
LIN {X 0,Y 587.27,Z 421.157,A -85,B 0,C 180,E1 -1459.577,E2 -1459.577} C_VEL
LIN {X 0,Y 587.321,Z 420.95,A -85,B 0,C 180,E1 -1461.774,E2 -1461.774} C_VEL
LIN {X 0,Y 587.346,Z 420.945,A -85,B 0,C 180,E1 -1464.759,E2 -1464.759} C_VEL
LIN {X 0,Y 587.325,Z 420.945,A -85,B 0,C 180,E1 -1467.046,E2 -1467.046} C_VEL
LIN {X 0,Y 587.347,Z 420.943,A -85,B 0,C 180,E1 -1469.379,E2 -1469.379} C_VEL
LIN {X 0,Y 587.353,Z 420.948,A -85,B 0,C 180,E1 -1471.838,E2 -1471.838} C_VEL
LIN {X 0,Y 587.351,Z 420.947,A -85,B 0,C 180,E1 -1474.35,E2 -1474.35} C_VEL
LIN {X 0,Y 587.348,Z 420.943,A -85,B 0,C 180,E1 -1476.747,E2 -1476.747} C_VEL
LIN {X 0,Y 587.342,Z 420.945,A -85,B 0,C 180,E1 -1479.36,E2 -1479.36} C_VEL
LIN {X 0,Y 587.33,Z 420.952,A -85,B 0,C 180,E1 -1482.108,E2 -1482.108} C_VEL
LIN {X 0,Y 587.312,Z 420.948,A -85,B 0,C 180,E1 -1484.912,E2 -1484.912} C_VEL
LIN {X 0,Y 587.35,Z 420.952,A -85,B 0,C 180,E1 -1487.928,E2 -1487.928} C_VEL
LIN {X 0,Y 587.388,Z 421.151,A -85,B 0,C 180,E1 -1490.534,E2 -1490.534} C_VEL
LIN {X 0,Y 587.74,Z 425.215,A -85,B 0,C 180,E1 -1492.111,E2 -1492.111} C_VEL
LIN {X 0,Y 587.626,Z 433.42,A -85,B 0,C 180,E1 -1494.966,E2 -1494.966} C_VEL
LIN {X 0,Y 587.588,Z 442.457,A -85,B 0,C 180,E1 -1497.821,E2 -1497.821} C_VEL
LIN {X 0,Y 587.521,Z 451.708,A -85,B 0,C 180,E1 -1500.631,E2 -1500.631} C_VEL
LIN {X 0,Y 587.489,Z 460.667,A -85,B 0,C 180,E1 -1503.346,E2 -1503.346} C_VEL
LIN {X 0,Y 587.385,Z 469.627,A -85,B 0,C 180,E1 -1505.996,E2 -1505.996} C_VEL
LIN {X 0,Y 587.348,Z 478.588,A -85,B 0,C 180,E1 -1508.596,E2 -1508.596} C_VEL
LIN {X 0,Y 587.299,Z 487.546,A -85,B 0,C 180,E1 -1511.15,E2 -1511.15} C_VEL
LIN {X 0,Y 587.259,Z 497.786,A -85,B 0,C 180,E1 -1514.023,E2 -1514.023} C_VEL
LIN {X 0,Y 587.258,Z 502.233,A -85,B 0,C 180,E1 -1515.258,E2 -1515.258} C_VEL
LIN {X 0,Y 588.012,Z 507.423,A -85,B 0,C 180,E1 -1515.357,E2 -1515.357} C_VEL
LIN {X 0,Y 587.938,Z 522.02,A -85,B 0,C 180,E1 -1515.66,E2 -1515.66} C_VEL
LIN {X 0,Y 587.825,Z 536.127,A -85,B 0,C 180,E1 -1516.103,E2 -1516.103} C_VEL
LIN {X 0,Y 587.742,Z 549.888,A -85,B 0,C 180,E1 -1516.692,E2 -1516.692} C_VEL
LIN {X 0,Y 587.624,Z 562.688,A -85,B 0,C 180,E1 -1517.393,E2 -1517.393} C_VEL
LIN {X 0,Y 587.513,Z 575.478,A -85,B 0,C 180,E1 -1518.267,E2 -1518.267} C_VEL
LIN {X 0,Y 587.467,Z 585.935,A -85,B 0,C 180,E1 -1519.14,E2 -1519.14} C_VEL
LIN {X 0,Y 587.353,Z 596.335,A -85,B 0,C 180,E1 -1520.183,E2 -1520.183} C_VEL
LIN {X 0,Y 587.311,Z 604.914,A -85,B 0,C 180,E1 -1521.224,E2 -1521.224} C_VEL
LIN {X 0,Y 587.249,Z 613.115,A -85,B 0,C 180,E1 -1522.436,E2 -1522.436} C_VEL
LIN {X 0,Y 587.179,Z 619.681,A -85,B 0,C 180,E1 -1523.635,E2 -1523.635} C_VEL
LIN {X 0,Y 587.16,Z 624.962,A -85,B 0,C 180,E1 -1524.85,E2 -1524.85} C_VEL
LIN {X 0,Y 587.179,Z 628.442,A -85,B 0,C 180,E1 -1525.882,E2 -1525.882} C_VEL
LIN {X 0,Y 587.13,Z 631.831,A -85,B 0,C 180,E1 -1527.256,E2 -1527.256} C_VEL
LIN {X 0,Y 587.141,Z 633.831,A -85,B 0,C 180,E1 -1528.628,E2 -1528.628} C_VEL
LIN {X 0,Y 587.135,Z 634.5,A -85,B 0,C 180,E1 -1530,E2 -1530} C_VEL
LIN {X 0,Y 587.141,Z 633.832,A -85,B 0,C 180,E1 -1531.372,E2 -1531.372} C_VEL
LIN {X 0,Y 587.13,Z 631.832,A -85,B 0,C 180,E1 -1532.744,E2 -1532.744} C_VEL
LIN {X 0,Y 587.179,Z 628.443,A -85,B 0,C 180,E1 -1534.118,E2 -1534.118} C_VEL
LIN {X 0,Y 587.199,Z 623.568,A -85,B 0,C 180,E1 -1535.494,E2 -1535.494} C_VEL
LIN {X 0,Y 587.209,Z 617.052,A -85,B 0,C 180,E1 -1536.874,E2 -1536.874} C_VEL
LIN {X 0,Y 587.268,Z 609.8,A -85,B 0,C 180,E1 -1538.083,E2 -1538.083} C_VEL
LIN {X 0,Y 587.321,Z 600.824,A -85,B 0,C 180,E1 -1539.296,E2 -1539.296} C_VEL
LIN {X 0,Y 587.372,Z 591.393,A -85,B 0,C 180,E1 -1540.339,E2 -1540.339} C_VEL
LIN {X 0,Y 587.474,Z 581.027,A -85,B 0,C 180,E1 -1541.29,E2 -1541.29} C_VEL
LIN {X 0,Y 587.578,Z 569.432,A -85,B 0,C 180,E1 -1542.17,E2 -1542.17} C_VEL
LIN {X 0,Y 587.666,Z 556.651,A -85,B 0,C 180,E1 -1542.958,E2 -1542.958} C_VEL
LIN {X 0,Y 587.789,Z 544.166,A -85,B 0,C 180,E1 -1543.571,E2 -1543.571} C_VEL
LIN {X 0,Y 587.896,Z 530.723,A -85,B 0,C 180,E1 -1544.082,E2 -1544.082} C_VEL
LIN {X 0,Y 587.943,Z 517.008,A -85,B 0,C 180,E1 -1544.46,E2 -1544.46} C_VEL
LIN {X 0,Y 587.84,Z 505.413,A -85,B 0,C 180,E1 -1544.677,E2 -1544.677} C_VEL
LIN {X 0,Y 587.268,Z 502.22,A -85,B 0,C 180,E1 -1544.745,E2 -1544.745} C_VEL
LIN {X 0,Y 587.303,Z 491.386,A -85,B 0,C 180,E1 -1547.767,E2 -1547.767} C_VEL
LIN {X 0,Y 587.344,Z 481.146,A -85,B 0,C 180,E1 -1550.67,E2 -1550.67} C_VEL
LIN {X 0,Y 587.395,Z 472.187,A -85,B 0,C 180,E1 -1553.255,E2 -1553.255} C_VEL
LIN {X 0,Y 587.458,Z 463.34,A -85,B 0,C 180,E1 -1555.857,E2 -1555.857} C_VEL
LIN {X 0,Y 587.501,Z 454.267,A -85,B 0,C 180,E1 -1558.587,E2 -1558.587} C_VEL
LIN {X 0,Y 587.578,Z 445.223,A -85,B 0,C 180,E1 -1561.352,E2 -1561.352} C_VEL
LIN {X 0,Y 587.661,Z 435.596,A -85,B 0,C 180,E1 -1564.392,E2 -1564.392} C_VEL
LIN {X 0,Y 587.731,Z 427.329,A -85,B 0,C 180,E1 -1567.146,E2 -1567.146} C_VEL
LIN {X 0,Y 587.576,Z 422.118,A -85,B 0,C 180,E1 -1568.971,E2 -1568.971} C_VEL
LIN {X 0,Y 587.341,Z 420.953,A -85,B 0,C 180,E1 -1569.47,E2 -1569.47} C_VEL
LIN {X 0,Y 587.331,Z 420.953,A -85,B 0,C 180,E1 -1572.107,E2 -1572.107} C_VEL
LIN {X 0,Y 587.313,Z 420.956,A -85,B 0,C 180,E1 -1575.088,E2 -1575.088} C_VEL
LIN {X 0,Y 587.348,Z 420.95,A -85,B 0,C 180,E1 -1577.927,E2 -1577.927} C_VEL
LIN {X 0,Y 587.329,Z 420.95,A -85,B 0,C 180,E1 -1581.058,E2 -1581.058} C_VEL
LIN {X 0,Y 587.35,Z 420.951,A -85,B 0,C 180,E1 -1583.291,E2 -1583.291} C_VEL
LIN {X 0,Y 587.359,Z 420.948,A -85,B 0,C 180,E1 -1585.78,E2 -1585.78} C_VEL
LIN {X 0,Y 587.35,Z 420.947,A -85,B 0,C 180,E1 -1588.232,E2 -1588.232} C_VEL
LIN {X 0,Y 587.349,Z 420.947,A -85,B 0,C 180,E1 -1590.865,E2 -1590.865} C_VEL
LIN {X 0,Y 587.36,Z 420.946,A -85,B 0,C 180,E1 -1593.817,E2 -1593.817} C_VEL
LIN {X 0,Y 587.317,Z 420.953,A -85,B 0,C 180,E1 -1596.741,E2 -1596.741} C_VEL
LIN {X 0,Y 587.329,Z 420.954,A -85,B 0,C 180,E1 -1599.695,E2 -1599.695} C_VEL
LIN {X 0,Y 587.353,Z 420.95,A -85,B 0,C 180,E1 -1602.594,E2 -1602.594} C_VEL
LIN {X 0,Y 587.358,Z 420.946,A -85,B 0,C 180,E1 -1605.739,E2 -1605.739} C_VEL
LIN {X 0,Y 587.355,Z 420.947,A -85,B 0,C 180,E1 -1608.859,E2 -1608.859} C_VEL
LIN {X 0,Y 587.367,Z 420.946,A -85,B 0,C 180,E1 -1611.745,E2 -1611.745} C_VEL
LIN {X 0,Y 587.358,Z 420.947,A -85,B 0,C 180,E1 -1614.507,E2 -1614.507} C_VEL
LIN {X 0,Y 587.374,Z 420.945,A -85,B 0,C 180,E1 -1617.257,E2 -1617.257} C_VEL
LIN {X 0,Y 587.375,Z 420.944,A -85,B 0,C 180,E1 -1620,E2 -1620} C_VEL
LIN {X 0,Y 587.378,Z 420.945,A -85,B 0,C 180,E1 -1622.743,E2 -1622.743} C_VEL
LIN {X 0,Y 587.363,Z 420.946,A -85,B 0,C 180,E1 -1625.493,E2 -1625.493} C_VEL
LIN {X 0,Y 587.366,Z 420.946,A -85,B 0,C 180,E1 -1628.255,E2 -1628.255} C_VEL
LIN {X 0,Y 587.34,Z 420.951,A -85,B 0,C 180,E1 -1631.134,E2 -1631.134} C_VEL
LIN {X 0,Y 587.354,Z 420.948,A -85,B 0,C 180,E1 -1633.846,E2 -1633.846} C_VEL
LIN {X 0,Y 587.36,Z 420.951,A -85,B 0,C 180,E1 -1636.821,E2 -1636.821} C_VEL
LIN {X 0,Y 587.32,Z 420.952,A -85,B 0,C 180,E1 -1638.325,E2 -1638.325} C_VEL
LIN {X 0,Y 586.667,Z 421.032,A -85,B 0,C 180,E1 -1638.897,E2 -1638.897} C_VEL
LIN {X 0,Y 583.838,Z 421.387,A -85,B 0,C 180,E1 -1639.825,E2 -1639.825} C_VEL
LIN {X 0,Y 581.429,Z 421.688,A -85,B 0,C 180,E1 -1640.572,E2 -1640.572} C_VEL
LIN {X 0,Y 580.377,Z 421.818,A -85,B 0,C 180,E1 -1641.149,E2 -1641.149} C_VEL
LIN {X 0,Y 580.282,Z 421.828,A -85,B 0,C 180,E1 -1641.344,E2 -1641.344} C_VEL
LIN {X 0,Y 580.297,Z 421.826,A -85,B 0,C 180,E1 -1644.317,E2 -1644.317} C_VEL
LIN {X 0,Y 580.273,Z 421.831,A -85,B 0,C 180,E1 -1646.624,E2 -1646.624} C_VEL
LIN {X 0,Y 580.298,Z 421.829,A -85,B 0,C 180,E1 -1649.311,E2 -1649.311} C_VEL
LIN {X 0,Y 580.3,Z 421.827,A -85,B 0,C 180,E1 -1652.201,E2 -1652.201} C_VEL
LIN {X 0,Y 580.288,Z 421.831,A -85,B 0,C 180,E1 -1654.697,E2 -1654.697} C_VEL
LIN {X 0,Y 580.298,Z 421.828,A -85,B 0,C 180,E1 -1657.269,E2 -1657.269} C_VEL
LIN {X 0,Y 580.29,Z 421.83,A -85,B 0,C 180,E1 -1660.271,E2 -1660.271} C_VEL
LIN {X 0,Y 580.29,Z 421.829,A -85,B 0,C 180,E1 -1662.706,E2 -1662.706} C_VEL
LIN {X 0,Y 580.272,Z 421.832,A -85,B 0,C 180,E1 -1665.609,E2 -1665.609} C_VEL
LIN {X 0,Y 580.279,Z 421.83,A -85,B 0,C 180,E1 -1668.232,E2 -1668.232} C_VEL
LIN {X 0,Y 580.289,Z 421.829,A -85,B 0,C 180,E1 -1670.967,E2 -1670.967} C_VEL
LIN {X 0,Y 580.297,Z 421.827,A -85,B 0,C 180,E1 -1673.599,E2 -1673.599} C_VEL
LIN {X 0,Y 580.322,Z 421.823,A -85,B 0,C 180,E1 -1676.146,E2 -1676.146} C_VEL
LIN {X 0,Y 580.278,Z 421.827,A -85,B 0,C 180,E1 -1678.615,E2 -1678.615} C_VEL
LIN {X 0,Y 580.295,Z 421.828,A -85,B 0,C 180,E1 -1681.025,E2 -1681.025} C_VEL
LIN {X 0,Y 580.295,Z 421.829,A -85,B 0,C 180,E1 -1683.666,E2 -1683.666} C_VEL
LIN {X 0,Y 580.303,Z 421.825,A -85,B 0,C 180,E1 -1685.684,E2 -1685.684} C_VEL
LIN {X 0,Y 580.276,Z 421.83,A -85,B 0,C 180,E1 -1687.948,E2 -1687.948} C_VEL
LIN {X 0,Y 580.303,Z 421.825,A -85,B 0,C 180,E1 -1690.914,E2 -1690.914} C_VEL
LIN {X 0,Y 580.28,Z 421.828,A -85,B 0,C 180,E1 -1693.826,E2 -1693.826} C_VEL
LIN {X 0,Y 580.33,Z 421.825,A -85,B 0,C 180,E1 -1695.983,E2 -1695.983} C_VEL
LIN {X 0,Y 580.31,Z 421.827,A -85,B 0,C 180,E1 -1698.827,E2 -1698.827} C_VEL
LIN {X 0,Y 580.333,Z 421.823,A -85,B 0,C 180,E1 -1701.644,E2 -1701.644} C_VEL
LIN {X 0,Y 580.325,Z 421.824,A -85,B 0,C 180,E1 -1704.44,E2 -1704.44} C_VEL
LIN {X 0,Y 580.339,Z 421.822,A -85,B 0,C 180,E1 -1707.224,E2 -1707.224} C_VEL
LIN {X 0,Y 580.357,Z 421.819,A -85,B 0,C 180,E1 -1710,E2 -1710} C_VEL
LIN {X 0,Y 580.341,Z 421.821,A -85,B 0,C 180,E1 -1712.776,E2 -1712.776} C_VEL
LIN {X 0,Y 580.331,Z 421.822,A -85,B 0,C 180,E1 -1715.56,E2 -1715.56} C_VEL
LIN {X 0,Y 580.328,Z 421.824,A -85,B 0,C 180,E1 -1717.655,E2 -1717.655} C_VEL
LIN {X 0,Y 580.307,Z 421.827,A -85,B 0,C 180,E1 -1720.466,E2 -1720.466} C_VEL
LIN {X 0,Y 580.276,Z 421.832,A -85,B 0,C 180,E1 -1723.304,E2 -1723.304} C_VEL
LIN {X 0,Y 580.296,Z 421.826,A -85,B 0,C 180,E1 -1725.452,E2 -1725.452} C_VEL
LIN {X 0,Y 580.293,Z 421.829,A -85,B 0,C 180,E1 -1727.624,E2 -1727.624} C_VEL
LIN {X 0,Y 580.29,Z 421.827,A -85,B 0,C 180,E1 -1729.822,E2 -1729.822} C_VEL
LIN {X 0,Y 580.272,Z 421.829,A -85,B 0,C 180,E1 -1732.052,E2 -1732.052} C_VEL
LIN {X 0,Y 580.31,Z 421.824,A -85,B 0,C 180,E1 -1735.079,E2 -1735.079} C_VEL
LIN {X 0,Y 580.305,Z 421.825,A -85,B 0,C 180,E1 -1738.185,E2 -1738.185} C_VEL
LIN {X 0,Y 580.295,Z 421.826,A -85,B 0,C 180,E1 -1740.695,E2 -1740.695} C_VEL
LIN {X 0,Y 580.282,Z 421.827,A -85,B 0,C 180,E1 -1743.312,E2 -1743.312} C_VEL
LIN {X 0,Y 580.205,Z 421.842,A -85,B 0,C 180,E1 -1744.701,E2 -1744.701} C_VEL
LIN {X 0,Y 580.156,Z 422.447,A -85,B 0,C 180,E1 -1745.743,E2 -1745.743} C_VEL
LIN {X 0,Y 580.135,Z 424.925,A -85,B 0,C 180,E1 -1748.157,E2 -1748.157} C_VEL
LIN {X 0,Y 580.11,Z 427.714,A -85,B 0,C 180,E1 -1750.859,E2 -1750.859} C_VEL
LIN {X 0,Y 580.119,Z 430.641,A -85,B 0,C 180,E1 -1753.672,E2 -1753.672} C_VEL
LIN {X 0,Y 580.09,Z 433.52,A -85,B 0,C 180,E1 -1756.324,E2 -1756.324} C_VEL
LIN {X 0,Y 580.07,Z 436.767,A -85,B 0,C 180,E1 -1759.137,E2 -1759.137} C_VEL
LIN {X 0,Y 580.059,Z 440.088,A -85,B 0,C 180,E1 -1761.955,E2 -1761.955} C_VEL
LIN {X 0,Y 580.057,Z 443.064,A -85,B 0,C 180,E1 -1764.439,E2 -1764.439} C_VEL
LIN {X 0,Y 580.068,Z 446.381,A -85,B 0,C 180,E1 -1767.167,E2 -1767.167} C_VEL
LIN {X 0,Y 581.114,Z 453.204,A -85,B 0,C 180,E1 -1767.33,E2 -1767.33} C_VEL
LIN {X 0,Y 581.007,Z 467.055,A -85,B 0,C 180,E1 -1767.677,E2 -1767.677} C_VEL
LIN {X 0,Y 580.89,Z 480.237,A -85,B 0,C 180,E1 -1768.142,E2 -1768.142} C_VEL
LIN {X 0,Y 580.788,Z 492.939,A -85,B 0,C 180,E1 -1768.73,E2 -1768.73} C_VEL
LIN {X 0,Y 580.634,Z 505.249,A -85,B 0,C 180,E1 -1769.445,E2 -1769.445} C_VEL
LIN {X 0,Y 580.541,Z 516.429,A -85,B 0,C 180,E1 -1770.241,E2 -1770.241} C_VEL
LIN {X 0,Y 580.417,Z 527.846,A -85,B 0,C 180,E1 -1771.228,E2 -1771.228} C_VEL
LIN {X 0,Y 580.297,Z 538.578,A -85,B 0,C 180,E1 -1772.369,E2 -1772.369} C_VEL
LIN {X 0,Y 580.2,Z 547.878,A -85,B 0,C 180,E1 -1773.578,E2 -1773.578} C_VEL
LIN {X 0,Y 580.147,Z 555.042,A -85,B 0,C 180,E1 -1774.721,E2 -1774.721} C_VEL
LIN {X 0,Y 580.127,Z 561.777,A -85,B 0,C 180,E1 -1776.056,E2 -1776.056} C_VEL
LIN {X 0,Y 580.1,Z 566.232,A -85,B 0,C 180,E1 -1777.189,E2 -1777.189} C_VEL
LIN {X 0,Y 580.068,Z 568.634,A -85,B 0,C 180,E1 -1777.939,E2 -1777.939} C_VEL
LIN {X 0,Y 580.062,Z 571.061,A -85,B 0,C 180,E1 -1778.893,E2 -1778.893} C_VEL
LIN {X 0,Y 580.027,Z 573.28,A -85,B 0,C 180,E1 -1780.168,E2 -1780.168} C_VEL
LIN {X 0,Y 580.032,Z 574.415,A -85,B 0,C 180,E1 -1781.637,E2 -1781.637} C_VEL
LIN {X 0,Y 580.029,Z 574.095,A -85,B 0,C 180,E1 -1783.094,E2 -1783.094} C_VEL
LIN {X 0,Y 580.036,Z 572.345,A -85,B 0,C 180,E1 -1784.54,E2 -1784.54} C_VEL
LIN {X 0,Y 580.078,Z 569.143,A -85,B 0,C 180,E1 -1785.977,E2 -1785.977} C_VEL
LIN {X 0,Y 580.096,Z 565.709,A -85,B 0,C 180,E1 -1787.048,E2 -1787.048} C_VEL
LIN {X 0,Y 580.112,Z 561.406,A -85,B 0,C 180,E1 -1788.115,E2 -1788.115} C_VEL
LIN {X 0,Y 580.167,Z 555.968,A -85,B 0,C 180,E1 -1789.208,E2 -1789.208} C_VEL
LIN {X 0,Y 580.204,Z 548.573,A -85,B 0,C 180,E1 -1790.412,E2 -1790.412} C_VEL
LIN {X 0,Y 580.256,Z 540.726,A -85,B 0,C 180,E1 -1791.467,E2 -1791.467} C_VEL
LIN {X 0,Y 580.37,Z 531.295,A -85,B 0,C 180,E1 -1792.52,E2 -1792.52} C_VEL
LIN {X 0,Y 580.486,Z 519.908,A -85,B 0,C 180,E1 -1793.567,E2 -1793.567} C_VEL
LIN {X 0,Y 580.612,Z 508.282,A -85,B 0,C 180,E1 -1794.443,E2 -1794.443} C_VEL
LIN {X 0,Y 580.767,Z 495.437,A -85,B 0,C 180,E1 -1795.228,E2 -1795.228} C_VEL
LIN {X 0,Y 580.878,Z 482.907,A -85,B 0,C 180,E1 -1795.837,E2 -1795.837} C_VEL
LIN {X 0,Y 581.002,Z 468.904,A -85,B 0,C 180,E1 -1796.359,E2 -1796.359} C_VEL
LIN {X 0,Y 581.091,Z 454.849,A -85,B 0,C 180,E1 -1796.728,E2 -1796.728} C_VEL
LIN {X 0,Y 580.812,Z 450.323,A -85,B 0,C 180,E1 -1796.824,E2 -1796.824} C_VEL
LIN {X 0,Y 580.052,Z 446.388,A -85,B 0,C 180,E1 -1796.918,E2 -1796.918} C_VEL
LIN {X 0,Y 580.078,Z 442.643,A -85,B 0,C 180,E1 -1800,E2 -1800} C_VEL
LIN {X 0,Y 580.052,Z 439.325,A -85,B 0,C 180,E1 -1802.778,E2 -1802.778} C_VEL
LIN {X 0,Y 580.11,Z 436.057,A -85,B 0,C 180,E1 -1805.562,E2 -1805.562} C_VEL
LIN {X 0,Y 580.108,Z 432.844,A -85,B 0,C 180,E1 -1808.359,E2 -1808.359} C_VEL
LIN {X 0,Y 580.085,Z 430.705,A -85,B 0,C 180,E1 -1810.471,E2 -1810.471} C_VEL
LIN {X 0,Y 580.139,Z 428.853,A -85,B 0,C 180,E1 -1812.595,E2 -1812.595} C_VEL
LIN {X 0,Y 580.166,Z 426.681,A -85,B 0,C 180,E1 -1814.737,E2 -1814.737} C_VEL
LIN {X 0,Y 580.216,Z 424.567,A -85,B 0,C 180,E1 -1816.9,E2 -1816.9} C_VEL
LIN {X 0,Y 580.23,Z 422.343,A -85,B 0,C 180,E1 -1819.134,E2 -1819.134} C_VEL
LIN {X 0,Y 580.215,Z 421.841,A -85,B 0,C 180,E1 -1819.825,E2 -1819.825} C_VEL
LIN {X 0,Y 580.272,Z 421.832,A -85,B 0,C 180,E1 -1822.053,E2 -1822.053} C_VEL
LIN {X 0,Y 580.303,Z 421.82,A -85,B 0,C 180,E1 -1825.08,E2 -1825.08} C_VEL
LIN {X 0,Y 580.314,Z 421.825,A -85,B 0,C 180,E1 -1827.864,E2 -1827.864} C_VEL
LIN {X 0,Y 580.294,Z 421.823,A -85,B 0,C 180,E1 -1830.698,E2 -1830.698} C_VEL
LIN {X 0,Y 580.301,Z 421.821,A -85,B 0,C 180,E1 -1833.317,E2 -1833.317} C_VEL
LIN {X 0,Y 580.321,Z 421.824,A -85,B 0,C 180,E1 -1835.768,E2 -1835.768} C_VEL
LIN {X 0,Y 580.285,Z 421.83,A -85,B 0,C 180,E1 -1838.147,E2 -1838.147} C_VEL
LIN {X 0,Y 580.297,Z 421.821,A -85,B 0,C 180,E1 -1840.844,E2 -1840.844} C_VEL
LIN {X 0,Y 580.285,Z 421.829,A -85,B 0,C 180,E1 -1843.657,E2 -1843.657} C_VEL
LIN {X 0,Y 580.282,Z 421.826,A -85,B 0,C 180,E1 -1846.609,E2 -1846.609} C_VEL
LIN {X 0,Y 580.298,Z 421.826,A -85,B 0,C 180,E1 -1849.157,E2 -1849.157} C_VEL
LIN {X 0,Y 580.293,Z 421.846,A -85,B 0,C 180,E1 -1850.165,E2 -1850.165} C_VEL
LIN {X 0,Y 580.786,Z 424.962,A -85,B 0,C 180,E1 -1851.452,E2 -1851.452} C_VEL
LIN {X 0,Y 580.712,Z 430.91,A -85,B 0,C 180,E1 -1853.629,E2 -1853.629} C_VEL
LIN {X 0,Y 580.595,Z 438.404,A -85,B 0,C 180,E1 -1856.164,E2 -1856.164} C_VEL
LIN {X 0,Y 580.575,Z 447.487,A -85,B 0,C 180,E1 -1858.987,E2 -1858.987} C_VEL
LIN {X 0,Y 580.506,Z 456.827,A -85,B 0,C 180,E1 -1861.826,E2 -1861.826} C_VEL
LIN {X 0,Y 580.436,Z 465.787,A -85,B 0,C 180,E1 -1864.543,E2 -1864.543} C_VEL
LIN {X 0,Y 580.336,Z 476.027,A -85,B 0,C 180,E1 -1867.576,E2 -1867.576} C_VEL
LIN {X 0,Y 580.281,Z 484.986,A -85,B 0,C 180,E1 -1870.177,E2 -1870.177} C_VEL
LIN {X 0,Y 580.229,Z 495.274,A -85,B 0,C 180,E1 -1873.114,E2 -1873.114} C_VEL
LIN {X 0,Y 580.173,Z 502.186,A -85,B 0,C 180,E1 -1875.061,E2 -1875.061} C_VEL
LIN {X 0,Y 581.159,Z 508.653,A -85,B 0,C 180,E1 -1875.199,E2 -1875.199} C_VEL
LIN {X 0,Y 581.052,Z 522.874,A -85,B 0,C 180,E1 -1875.51,E2 -1875.51} C_VEL
LIN {X 0,Y 580.937,Z 536.241,A -85,B 0,C 180,E1 -1875.94,E2 -1875.94} C_VEL
LIN {X 0,Y 580.836,Z 549.887,A -85,B 0,C 180,E1 -1876.531,E2 -1876.531} C_VEL
LIN {X 0,Y 580.664,Z 562.689,A -85,B 0,C 180,E1 -1877.239,E2 -1877.239} C_VEL
LIN {X 0,Y 580.544,Z 575.479,A -85,B 0,C 180,E1 -1878.124,E2 -1878.124} C_VEL
LIN {X 0,Y 580.461,Z 585.974,A -85,B 0,C 180,E1 -1879.01,E2 -1879.01} C_VEL
LIN {X 0,Y 580.311,Z 596.335,A -85,B 0,C 180,E1 -1880.062,E2 -1880.062} C_VEL
LIN {X 0,Y 580.254,Z 604.914,A -85,B 0,C 180,E1 -1881.117,E2 -1881.117} C_VEL
LIN {X 0,Y 580.176,Z 613.116,A -85,B 0,C 180,E1 -1882.343,E2 -1882.343} C_VEL
LIN {X 0,Y 580.123,Z 618.992,A -85,B 0,C 180,E1 -1883.416,E2 -1883.416} C_VEL
LIN {X 0,Y 580.128,Z 623.569,A -85,B 0,C 180,E1 -1884.438,E2 -1884.438} C_VEL
LIN {X 0,Y 580.102,Z 628.443,A -85,B 0,C 180,E1 -1885.832,E2 -1885.832} C_VEL
LIN {X 0,Y 580.041,Z 631.832,A -85,B 0,C 180,E1 -1887.222,E2 -1887.222} C_VEL
LIN {X 0,Y 580.041,Z 633.832,A -85,B 0,C 180,E1 -1888.611,E2 -1888.611} C_VEL
LIN {X 0,Y 580.036,Z 634.5,A -85,B 0,C 180,E1 -1890,E2 -1890} C_VEL
LIN {X 0,Y 580.041,Z 633.832,A -85,B 0,C 180,E1 -1891.389,E2 -1891.389} C_VEL
LIN {X 0,Y 580.041,Z 631.833,A -85,B 0,C 180,E1 -1892.778,E2 -1892.778} C_VEL
LIN {X 0,Y 580.102,Z 628.444,A -85,B 0,C 180,E1 -1894.168,E2 -1894.168} C_VEL
LIN {X 0,Y 580.128,Z 623.568,A -85,B 0,C 180,E1 -1895.562,E2 -1895.562} C_VEL
LIN {X 0,Y 580.141,Z 617.053,A -85,B 0,C 180,E1 -1896.958,E2 -1896.958} C_VEL
LIN {X 0,Y 580.192,Z 609.8,A -85,B 0,C 180,E1 -1898.183,E2 -1898.183} C_VEL
LIN {X 0,Y 580.283,Z 600.824,A -85,B 0,C 180,E1 -1899.41,E2 -1899.41} C_VEL
LIN {X 0,Y 580.356,Z 591.393,A -85,B 0,C 180,E1 -1900.466,E2 -1900.466} C_VEL
LIN {X 0,Y 580.475,Z 581.32,A -85,B 0,C 180,E1 -1901.404,E2 -1901.404} C_VEL
LIN {X 0,Y 580.592,Z 569.434,A -85,B 0,C 180,E1 -1902.318,E2 -1902.318} C_VEL
LIN {X 0,Y 580.726,Z 556.652,A -85,B 0,C 180,E1 -1903.115,E2 -1903.115} C_VEL
LIN {X 0,Y 580.865,Z 544.165,A -85,B 0,C 180,E1 -1903.736,E2 -1903.736} C_VEL
LIN {X 0,Y 581.009,Z 531.234,A -85,B 0,C 180,E1 -1904.234,E2 -1904.234} C_VEL
LIN {X 0,Y 581.077,Z 517.282,A -85,B 0,C 180,E1 -1904.628,E2 -1904.628} C_VEL
LIN {X 0,Y 580.961,Z 506.231,A -85,B 0,C 180,E1 -1904.842,E2 -1904.842} C_VEL
LIN {X 0,Y 580.178,Z 502.186,A -85,B 0,C 180,E1 -1904.939,E2 -1904.939} C_VEL
LIN {X 0,Y 580.234,Z 492.666,A -85,B 0,C 180,E1 -1907.626,E2 -1907.626} C_VEL
LIN {X 0,Y 580.289,Z 482.426,A -85,B 0,C 180,E1 -1910.562,E2 -1910.562} C_VEL
LIN {X 0,Y 580.337,Z 474.003,A -85,B 0,C 180,E1 -1913.019,E2 -1913.019} C_VEL
LIN {X 0,Y 580.436,Z 465.787,A -85,B 0,C 180,E1 -1915.457,E2 -1915.457} C_VEL
LIN {X 0,Y 580.506,Z 456.827,A -85,B 0,C 180,E1 -1918.174,E2 -1918.174} C_VEL
LIN {X 0,Y 580.578,Z 447.566,A -85,B 0,C 180,E1 -1921.015,E2 -1921.015} C_VEL
LIN {X 0,Y 580.611,Z 440.12,A -85,B 0,C 180,E1 -1923.362,E2 -1923.362} C_VEL
LIN {X 0,Y 580.723,Z 432.71,A -85,B 0,C 180,E1 -1925.821,E2 -1925.821} C_VEL
LIN {X 0,Y 580.805,Z 425.987,A -85,B 0,C 180,E1 -1928.138,E2 -1928.138} C_VEL
LIN {X 0,Y 580.319,Z 421.827,A -85,B 0,C 180,E1 -1929.686,E2 -1929.686} C_VEL
LIN {X 0,Y 580.276,Z 421.83,A -85,B 0,C 180,E1 -1932.706,E2 -1932.706} C_VEL
LIN {X 0,Y 580.27,Z 421.829,A -85,B 0,C 180,E1 -1935.608,E2 -1935.608} C_VEL
LIN {X 0,Y 580.31,Z 421.824,A -85,B 0,C 180,E1 -1938.234,E2 -1938.234} C_VEL
LIN {X 0,Y 580.284,Z 421.828,A -85,B 0,C 180,E1 -1940.966,E2 -1940.966} C_VEL
LIN {X 0,Y 580.278,Z 421.829,A -85,B 0,C 180,E1 -1943.597,E2 -1943.597} C_VEL
LIN {X 0,Y 580.314,Z 421.827,A -85,B 0,C 180,E1 -1946.145,E2 -1946.145} C_VEL
LIN {X 0,Y 580.286,Z 421.83,A -85,B 0,C 180,E1 -1948.615,E2 -1948.615} C_VEL
LIN {X 0,Y 580.293,Z 421.827,A -85,B 0,C 180,E1 -1951.024,E2 -1951.024} C_VEL
LIN {X 0,Y 580.325,Z 421.822,A -85,B 0,C 180,E1 -1953.657,E2 -1953.657} C_VEL
LIN {X 0,Y 580.274,Z 421.828,A -85,B 0,C 180,E1 -1956.442,E2 -1956.442} C_VEL
LIN {X 0,Y 580.278,Z 421.829,A -85,B 0,C 180,E1 -1959.437,E2 -1959.437} C_VEL
LIN {X 0,Y 580.276,Z 421.828,A -85,B 0,C 180,E1 -1961.645,E2 -1961.645} C_VEL
LIN {X 0,Y 580.28,Z 421.832,A -85,B 0,C 180,E1 -1963.826,E2 -1963.826} C_VEL
LIN {X 0,Y 580.319,Z 421.822,A -85,B 0,C 180,E1 -1965.983,E2 -1965.983} C_VEL
LIN {X 0,Y 580.325,Z 421.822,A -85,B 0,C 180,E1 -1968.827,E2 -1968.827} C_VEL
LIN {X 0,Y 580.331,Z 421.822,A -85,B 0,C 180,E1 -1971.644,E2 -1971.644} C_VEL
LIN {X 0,Y 580.323,Z 421.823,A -85,B 0,C 180,E1 -1974.44,E2 -1974.44} C_VEL
LIN {X 0,Y 580.34,Z 421.821,A -85,B 0,C 180,E1 -1977.224,E2 -1977.224} C_VEL
LIN {X 0,Y 580.345,Z 421.82,A -85,B 0,C 180,E1 -1980,E2 -1980} C_VEL
LIN {X 0,Y 580.343,Z 421.821,A -85,B 0,C 180,E1 -1982.777,E2 -1982.777} C_VEL
LIN {X 0,Y 580.33,Z 421.823,A -85,B 0,C 180,E1 -1985.56,E2 -1985.56} C_VEL
LIN {X 0,Y 580.329,Z 421.823,A -85,B 0,C 180,E1 -1988.356,E2 -1988.356} C_VEL
LIN {X 0,Y 580.292,Z 421.829,A -85,B 0,C 180,E1 -1991.191,E2 -1991.191} C_VEL
LIN {X 0,Y 580.32,Z 421.826,A -85,B 0,C 180,E1 -1994.017,E2 -1994.017} C_VEL
LIN {X 0,Y 580.31,Z 421.828,A -85,B 0,C 180,E1 -1996.916,E2 -1996.916} C_VEL
LIN {X 0,Y 580.303,Z 421.827,A -85,B 0,C 180,E1 -1999.823,E2 -1999.823} C_VEL
LIN {X 0,Y 580.282,Z 421.828,A -85,B 0,C 180,E1 -2001.344,E2 -2001.344} C_VEL
LIN {X 0,Y 579.585,Z 421.916,A -85,B 0,C 180,E1 -2001.923,E2 -2001.923} C_VEL
LIN {X 0,Y 576.708,Z 422.273,A -85,B 0,C 180,E1 -2002.863,E2 -2002.863} C_VEL
LIN {X 0,Y 574.312,Z 422.574,A -85,B 0,C 180,E1 -2003.619,E2 -2003.619} C_VEL
LIN {X 0,Y 573.314,Z 422.696,A -85,B 0,C 180,E1 -2004.203,E2 -2004.203} C_VEL
LIN {X 0,Y 573.247,Z 422.704,A -85,B 0,C 180,E1 -2004.401,E2 -2004.401} C_VEL
LIN {X 0,Y 573.247,Z 422.704,A -85,B 0,C 180,E1 -2006.976,E2 -2006.976} C_VEL
LIN {X 0,Y 573.243,Z 422.706,A -85,B 0,C 180,E1 -2009.489,E2 -2009.489} C_VEL
LIN {X 0,Y 573.253,Z 422.705,A -85,B 0,C 180,E1 -2012.23,E2 -2012.23} C_VEL
LIN {X 0,Y 573.238,Z 422.708,A -85,B 0,C 180,E1 -2014.773,E2 -2014.773} C_VEL
LIN {X 0,Y 573.251,Z 422.705,A -85,B 0,C 180,E1 -2017.167,E2 -2017.167} C_VEL
LIN {X 0,Y 573.237,Z 422.705,A -85,B 0,C 180,E1 -2019.608,E2 -2019.608} C_VEL
LIN {X 0,Y 573.249,Z 422.705,A -85,B 0,C 180,E1 -2022.644,E2 -2022.644} C_VEL
LIN {X 0,Y 573.238,Z 422.709,A -85,B 0,C 180,E1 -2025.668,E2 -2025.668} C_VEL
LIN {X 0,Y 573.229,Z 422.709,A -85,B 0,C 180,E1 -2028.544,E2 -2028.544} C_VEL
LIN {X 0,Y 573.248,Z 422.707,A -85,B 0,C 180,E1 -2031.3,E2 -2031.3} C_VEL
LIN {X 0,Y 573.265,Z 422.705,A -85,B 0,C 180,E1 -2034.012,E2 -2034.012} C_VEL
LIN {X 0,Y 573.286,Z 422.702,A -85,B 0,C 180,E1 -2036.52,E2 -2036.52} C_VEL
LIN {X 0,Y 573.235,Z 422.706,A -85,B 0,C 180,E1 -2039.117,E2 -2039.117} C_VEL
LIN {X 0,Y 573.239,Z 422.705,A -85,B 0,C 180,E1 -2041.436,E2 -2041.436} C_VEL
LIN {X 0,Y 573.268,Z 422.703,A -85,B 0,C 180,E1 -2043.811,E2 -2043.811} C_VEL
LIN {X 0,Y 573.234,Z 422.708,A -85,B 0,C 180,E1 -2046.135,E2 -2046.135} C_VEL
LIN {X 0,Y 573.253,Z 422.707,A -85,B 0,C 180,E1 -2049.174,E2 -2049.174} C_VEL
LIN {X 0,Y 573.225,Z 422.707,A -85,B 0,C 180,E1 -2051.412,E2 -2051.412} C_VEL
LIN {X 0,Y 573.252,Z 422.704,A -85,B 0,C 180,E1 -2053.622,E2 -2053.622} C_VEL
LIN {X 0,Y 573.277,Z 422.703,A -85,B 0,C 180,E1 -2055.807,E2 -2055.807} C_VEL
LIN {X 0,Y 573.267,Z 422.705,A -85,B 0,C 180,E1 -2058.745,E2 -2058.745} C_VEL
LIN {X 0,Y 573.288,Z 422.702,A -85,B 0,C 180,E1 -2061.541,E2 -2061.541} C_VEL
LIN {X 0,Y 573.292,Z 422.701,A -85,B 0,C 180,E1 -2064.372,E2 -2064.372} C_VEL
LIN {X 0,Y 573.316,Z 422.696,A -85,B 0,C 180,E1 -2067.892,E2 -2067.892} C_VEL
LIN {X 0,Y 573.331,Z 422.694,A -85,B 0,C 180,E1 -2070.702,E2 -2070.702} C_VEL
LIN {X 0,Y 573.308,Z 422.697,A -85,B 0,C 180,E1 -2072.811,E2 -2072.811} C_VEL
LIN {X 0,Y 573.298,Z 422.698,A -85,B 0,C 180,E1 -2075.628,E2 -2075.628} C_VEL
LIN {X 0,Y 573.276,Z 422.703,A -85,B 0,C 180,E1 -2077.75,E2 -2077.75} C_VEL
LIN {X 0,Y 573.273,Z 422.704,A -85,B 0,C 180,E1 -2080.596,E2 -2080.596} C_VEL
LIN {X 0,Y 573.267,Z 422.701,A -85,B 0,C 180,E1 -2082.748,E2 -2082.748} C_VEL
LIN {X 0,Y 573.239,Z 422.708,A -85,B 0,C 180,E1 -2084.919,E2 -2084.919} C_VEL
LIN {X 0,Y 573.245,Z 422.705,A -85,B 0,C 180,E1 -2087.848,E2 -2087.848} C_VEL
LIN {X 0,Y 573.245,Z 422.706,A -85,B 0,C 180,E1 -2090.076,E2 -2090.076} C_VEL
LIN {X 0,Y 573.238,Z 422.704,A -85,B 0,C 180,E1 -2092.337,E2 -2092.337} C_VEL
LIN {X 0,Y 573.257,Z 422.704,A -85,B 0,C 180,E1 -2095.409,E2 -2095.409} C_VEL
LIN {X 0,Y 573.267,Z 422.701,A -85,B 0,C 180,E1 -2098.031,E2 -2098.031} C_VEL
LIN {X 0,Y 573.241,Z 422.705,A -85,B 0,C 180,E1 -2100.883,E2 -2100.883} C_VEL
LIN {X 0,Y 573.241,Z 422.705,A -85,B 0,C 180,E1 -2103.52,E2 -2103.52} C_VEL
LIN {X 0,Y 573.089,Z 422.729,A -85,B 0,C 180,E1 -2105.195,E2 -2105.195} C_VEL
LIN {X 0,Y 573.068,Z 424.483,A -85,B 0,C 180,E1 -2107.141,E2 -2107.141} C_VEL
LIN {X 0,Y 573.039,Z 427.018,A -85,B 0,C 180,E1 -2109.623,E2 -2109.623} C_VEL
LIN {X 0,Y 573.016,Z 430.095,A -85,B 0,C 180,E1 -2112.617,E2 -2112.617} C_VEL
LIN {X 0,Y 573.031,Z 432.872,A -85,B 0,C 180,E1 -2115.344,E2 -2115.344} C_VEL
LIN {X 0,Y 573,Z 436.301,A -85,B 0,C 180,E1 -2118.432,E2 -2118.432} C_VEL
LIN {X 0,Y 572.958,Z 439.596,A -85,B 0,C 180,E1 -2121.275,E2 -2121.275} C_VEL
LIN {X 0,Y 572.925,Z 442.879,A -85,B 0,C 180,E1 -2124.057,E2 -2124.057} C_VEL
LIN {X 0,Y 572.973,Z 446.391,A -85,B 0,C 180,E1 -2126.987,E2 -2126.987} C_VEL
LIN {X 0,Y 574.252,Z 453.324,A -85,B 0,C 180,E1 -2127.153,E2 -2127.153} C_VEL
LIN {X 0,Y 574.131,Z 467.712,A -85,B 0,C 180,E1 -2127.52,E2 -2127.52} C_VEL
LIN {X 0,Y 573.975,Z 481.139,A -85,B 0,C 180,E1 -2128.008,E2 -2128.008} C_VEL
LIN {X 0,Y 573.853,Z 493.958,A -85,B 0,C 180,E1 -2128.619,E2 -2128.619} C_VEL
LIN {X 0,Y 573.684,Z 506.046,A -85,B 0,C 180,E1 -2129.34,E2 -2129.34} C_VEL
LIN {X 0,Y 573.544,Z 517.673,A -85,B 0,C 180,E1 -2130.194,E2 -2130.194} C_VEL
LIN {X 0,Y 573.392,Z 528.334,A -85,B 0,C 180,E1 -2131.143,E2 -2131.143} C_VEL
LIN {X 0,Y 573.242,Z 538.44,A -85,B 0,C 180,E1 -2132.232,E2 -2132.232} C_VEL
LIN {X 0,Y 573.188,Z 546.722,A -85,B 0,C 180,E1 -2133.308,E2 -2133.308} C_VEL
LIN {X 0,Y 573.063,Z 554.762,A -85,B 0,C 180,E1 -2134.581,E2 -2134.581} C_VEL
LIN {X 0,Y 573.045,Z 560.679,A -85,B 0,C 180,E1 -2135.741,E2 -2135.741} C_VEL
LIN {X 0,Y 573.013,Z 565.447,A -85,B 0,C 180,E1 -2136.905,E2 -2136.905} C_VEL
LIN {X 0,Y 572.989,Z 569.056,A -85,B 0,C 180,E1 -2138.031,E2 -2138.031} C_VEL
LIN {X 0,Y 572.96,Z 571.69,A -85,B 0,C 180,E1 -2139.162,E2 -2139.162} C_VEL
LIN {X 0,Y 572.934,Z 573.854,A -85,B 0,C 180,E1 -2140.658,E2 -2140.658} C_VEL
LIN {X 0,Y 572.938,Z 574.485,A -85,B 0,C 180,E1 -2142.141,E2 -2142.141} C_VEL
LIN {X 0,Y 572.934,Z 573.653,A -85,B 0,C 180,E1 -2143.612,E2 -2143.612} C_VEL
LIN {X 0,Y 572.952,Z 571.393,A -85,B 0,C 180,E1 -2145.073,E2 -2145.073} C_VEL
LIN {X 0,Y 573.008,Z 567.665,A -85,B 0,C 180,E1 -2146.524,E2 -2146.524} C_VEL
LIN {X 0,Y 573.03,Z 562.401,A -85,B 0,C 180,E1 -2147.965,E2 -2147.965} C_VEL
LIN {X 0,Y 573.08,Z 556.883,A -85,B 0,C 180,E1 -2149.122,E2 -2149.122} C_VEL
LIN {X 0,Y 573.141,Z 548.884,A -85,B 0,C 180,E1 -2150.471,E2 -2150.471} C_VEL
LIN {X 0,Y 573.212,Z 541.09,A -85,B 0,C 180,E1 -2151.539,E2 -2151.539} C_VEL
LIN {X 0,Y 573.359,Z 531.737,A -85,B 0,C 180,E1 -2152.605,E2 -2152.605} C_VEL
LIN {X 0,Y 573.477,Z 520.405,A -85,B 0,C 180,E1 -2153.667,E2 -2153.667} C_VEL
LIN {X 0,Y 573.626,Z 508.926,A -85,B 0,C 180,E1 -2154.551,E2 -2154.551} C_VEL
LIN {X 0,Y 573.815,Z 496.217,A -85,B 0,C 180,E1 -2155.346,E2 -2155.346} C_VEL
LIN {X 0,Y 573.946,Z 483.882,A -85,B 0,C 180,E1 -2155.962,E2 -2155.962} C_VEL
LIN {X 0,Y 574.101,Z 470.195,A -85,B 0,C 180,E1 -2156.491,E2 -2156.491} C_VEL
LIN {X 0,Y 574.232,Z 455.86,A -85,B 0,C 180,E1 -2156.887,E2 -2156.887} C_VEL
LIN {X 0,Y 573.946,Z 451.393,A -85,B 0,C 180,E1 -2156.984,E2 -2156.984} C_VEL
LIN {X 0,Y 572.951,Z 446.396,A -85,B 0,C 180,E1 -2157.1,E2 -2157.1} C_VEL
LIN {X 0,Y 572.984,Z 442.917,A -85,B 0,C 180,E1 -2160,E2 -2160} C_VEL
LIN {X 0,Y 572.965,Z 439.599,A -85,B 0,C 180,E1 -2162.812,E2 -2162.812} C_VEL
LIN {X 0,Y 573.033,Z 436.331,A -85,B 0,C 180,E1 -2165.631,E2 -2165.631} C_VEL
LIN {X 0,Y 573.034,Z 433.192,A -85,B 0,C 180,E1 -2168.463,E2 -2168.463} C_VEL
LIN {X 0,Y 573.097,Z 430.739,A -85,B 0,C 180,E1 -2171.315,E2 -2171.315} C_VEL
LIN {X 0,Y 573.121,Z 427.719,A -85,B 0,C 180,E1 -2174.365,E2 -2174.365} C_VEL
LIN {X 0,Y 573.16,Z 425.108,A -85,B 0,C 180,E1 -2177.115,E2 -2177.115} C_VEL
LIN {X 0,Y 573.171,Z 422.919,A -85,B 0,C 180,E1 -2179.333,E2 -2179.333} C_VEL
LIN {X 0,Y 573.227,Z 422.704,A -85,B 0,C 180,E1 -2181.581,E2 -2181.581} C_VEL
LIN {X 0,Y 573.269,Z 422.7,A -85,B 0,C 180,E1 -2184.634,E2 -2184.634} C_VEL
LIN {X 0,Y 573.259,Z 422.698,A -85,B 0,C 180,E1 -2186.975,E2 -2186.975} C_VEL
LIN {X 0,Y 573.248,Z 422.701,A -85,B 0,C 180,E1 -2189.49,E2 -2189.49} C_VEL
LIN {X 0,Y 573.252,Z 422.706,A -85,B 0,C 180,E1 -2192.23,E2 -2192.23} C_VEL
LIN {X 0,Y 573.246,Z 422.7,A -85,B 0,C 180,E1 -2194.774,E2 -2194.774} C_VEL
LIN {X 0,Y 573.25,Z 422.699,A -85,B 0,C 180,E1 -2197.167,E2 -2197.167} C_VEL
LIN {X 0,Y 573.244,Z 422.705,A -85,B 0,C 180,E1 -2199.607,E2 -2199.607} C_VEL
LIN {X 0,Y 573.24,Z 422.702,A -85,B 0,C 180,E1 -2202.643,E2 -2202.643} C_VEL
LIN {X 0,Y 573.236,Z 422.71,A -85,B 0,C 180,E1 -2205.668,E2 -2205.668} C_VEL
LIN {X 0,Y 573.242,Z 422.706,A -85,B 0,C 180,E1 -2208.545,E2 -2208.545} C_VEL
LIN {X 0,Y 573.276,Z 422.894,A -85,B 0,C 180,E1 -2209.939,E2 -2209.939} C_VEL
LIN {X 0,Y 573.828,Z 426.884,A -85,B 0,C 180,E1 -2211.614,E2 -2211.614} C_VEL
LIN {X 0,Y 573.703,Z 433.295,A -85,B 0,C 180,E1 -2213.985,E2 -2213.985} C_VEL
LIN {X 0,Y 573.58,Z 440.773,A -85,B 0,C 180,E1 -2216.539,E2 -2216.539} C_VEL
LIN {X 0,Y 573.568,Z 448.93,A -85,B 0,C 180,E1 -2219.061,E2 -2219.061} C_VEL
LIN {X 0,Y 573.49,Z 458.297,A -85,B 0,C 180,E1 -2221.927,E2 -2221.927} C_VEL
LIN {X 0,Y 573.412,Z 467.067,A -85,B 0,C 180,E1 -2224.598,E2 -2224.598} C_VEL
LIN {X 0,Y 573.322,Z 477.307,A -85,B 0,C 180,E1 -2227.666,E2 -2227.666} C_VEL
LIN {X 0,Y 573.232,Z 487.546,A -85,B 0,C 180,E1 -2230.669,E2 -2230.669} C_VEL
LIN {X 0,Y 573.156,Z 497.786,A -85,B 0,C 180,E1 -2233.619,E2 -2233.619} C_VEL
LIN {X 0,Y 573.132,Z 502.186,A -85,B 0,C 180,E1 -2234.873,E2 -2234.873} C_VEL
LIN {X 0,Y 574.305,Z 508.653,A -85,B 0,C 180,E1 -2235.018,E2 -2235.018} C_VEL
LIN {X 0,Y 574.172,Z 523.363,A -85,B 0,C 180,E1 -2235.347,E2 -2235.347} C_VEL
LIN {X 0,Y 573.997,Z 537.718,A -85,B 0,C 180,E1 -2235.826,E2 -2235.826} C_VEL
LIN {X 0,Y 573.881,Z 551.645,A -85,B 0,C 180,E1 -2236.455,E2 -2236.455} C_VEL
LIN {X 0,Y 573.705,Z 564.102,A -85,B 0,C 180,E1 -2237.172,E2 -2237.172} C_VEL
LIN {X 0,Y 573.572,Z 575.481,A -85,B 0,C 180,E1 -2237.977,E2 -2237.977} C_VEL
LIN {X 0,Y 573.449,Z 586.85,A -85,B 0,C 180,E1 -2238.955,E2 -2238.955} C_VEL
LIN {X 0,Y 573.268,Z 596.335,A -85,B 0,C 180,E1 -2239.939,E2 -2239.939} C_VEL
LIN {X 0,Y 573.19,Z 604.914,A -85,B 0,C 180,E1 -2241.006,E2 -2241.006} C_VEL
LIN {X 0,Y 573.111,Z 613.116,A -85,B 0,C 180,E1 -2242.248,E2 -2242.248} C_VEL
LIN {X 0,Y 573.035,Z 619.45,A -85,B 0,C 180,E1 -2243.427,E2 -2243.427} C_VEL
LIN {X 0,Y 573.001,Z 624.961,A -85,B 0,C 180,E1 -2244.722,E2 -2244.722} C_VEL
LIN {X 0,Y 573.028,Z 628.443,A -85,B 0,C 180,E1 -2245.78,E2 -2245.78} C_VEL
LIN {X 0,Y 572.956,Z 631.832,A -85,B 0,C 180,E1 -2247.188,E2 -2247.188} C_VEL
LIN {X 0,Y 572.941,Z 633.832,A -85,B 0,C 180,E1 -2248.594,E2 -2248.594} C_VEL
LIN {X 0,Y 572.937,Z 634.5,A -85,B 0,C 180,E1 -2250,E2 -2250} C_VEL
LIN {X 0,Y 572.941,Z 633.833,A -85,B 0,C 180,E1 -2251.406,E2 -2251.406} C_VEL
LIN {X 0,Y 572.956,Z 631.833,A -85,B 0,C 180,E1 -2252.812,E2 -2252.812} C_VEL
LIN {X 0,Y 573.028,Z 628.444,A -85,B 0,C 180,E1 -2254.22,E2 -2254.22} C_VEL
LIN {X 0,Y 573.059,Z 623.568,A -85,B 0,C 180,E1 -2255.63,E2 -2255.63} C_VEL
LIN {X 0,Y 573.058,Z 618.852,A -85,B 0,C 180,E1 -2256.693,E2 -2256.693} C_VEL
LIN {X 0,Y 573.126,Z 612.039,A -85,B 0,C 180,E1 -2257.929,E2 -2257.929} C_VEL
LIN {X 0,Y 573.225,Z 603.56,A -85,B 0,C 180,E1 -2259.171,E2 -2259.171} C_VEL
LIN {X 0,Y 573.304,Z 594.709,A -85,B 0,C 180,E1 -2260.239,E2 -2260.239} C_VEL
LIN {X 0,Y 573.461,Z 583.994,A -85,B 0,C 180,E1 -2261.308,E2 -2261.308} C_VEL
LIN {X 0,Y 573.621,Z 573.147,A -85,B 0,C 180,E1 -2262.201,E2 -2262.201} C_VEL
LIN {X 0,Y 573.735,Z 561.263,A -85,B 0,C 180,E1 -2263.008,E2 -2263.008} C_VEL
LIN {X 0,Y 573.949,Z 548.1,A -85,B 0,C 180,E1 -2263.724,E2 -2263.724} C_VEL
LIN {X 0,Y 574.073,Z 534.882,A -85,B 0,C 180,E1 -2264.283,E2 -2264.283} C_VEL
LIN {X 0,Y 574.195,Z 520.913,A -85,B 0,C 180,E1 -2264.718,E2 -2264.718} C_VEL
LIN {X 0,Y 574.172,Z 507.528,A -85,B 0,C 180,E1 -2265.002,E2 -2265.002} C_VEL
LIN {X 0,Y 573.134,Z 502.186,A -85,B 0,C 180,E1 -2265.127,E2 -2265.127} C_VEL
LIN {X 0,Y 573.182,Z 492.666,A -85,B 0,C 180,E1 -2267.85,E2 -2267.85} C_VEL
LIN {X 0,Y 573.24,Z 483.706,A -85,B 0,C 180,E1 -2270.451,E2 -2270.451} C_VEL
LIN {X 0,Y 573.312,Z 474.524,A -85,B 0,C 180,E1 -2273.162,E2 -2273.162} C_VEL
LIN {X 0,Y 573.416,Z 465.787,A -85,B 0,C 180,E1 -2275.791,E2 -2275.791} C_VEL
LIN {X 0,Y 573.492,Z 456.765,A -85,B 0,C 180,E1 -2278.55,E2 -2278.55} C_VEL
LIN {X 0,Y 573.61,Z 447.647,A -85,B 0,C 180,E1 -2281.38,E2 -2281.38} C_VEL
LIN {X 0,Y 573.703,Z 438.659,A -85,B 0,C 180,E1 -2284.298,E2 -2284.298} C_VEL
LIN {X 0,Y 573.829,Z 430.023,A -85,B 0,C 180,E1 -2287.242,E2 -2287.242} C_VEL
LIN {X 0,Y 573.703,Z 425.001,A -85,B 0,C 180,E1 -2289.053,E2 -2289.053} C_VEL
LIN {X 0,Y 573.259,Z 422.706,A -85,B 0,C 180,E1 -2289.948,E2 -2289.948} C_VEL
LIN {X 0,Y 573.238,Z 422.707,A -85,B 0,C 180,E1 -2292.641,E2 -2292.641} C_VEL
LIN {X 0,Y 573.236,Z 422.705,A -85,B 0,C 180,E1 -2295.667,E2 -2295.667} C_VEL
LIN {X 0,Y 573.241,Z 422.704,A -85,B 0,C 180,E1 -2298.544,E2 -2298.544} C_VEL
LIN {X 0,Y 573.244,Z 422.704,A -85,B 0,C 180,E1 -2301.299,E2 -2301.299} C_VEL
LIN {X 0,Y 573.24,Z 422.704,A -85,B 0,C 180,E1 -2304.013,E2 -2304.013} C_VEL
LIN {X 0,Y 573.279,Z 422.7,A -85,B 0,C 180,E1 -2306.519,E2 -2306.519} C_VEL
LIN {X 0,Y 573.239,Z 422.706,A -85,B 0,C 180,E1 -2309.115,E2 -2309.115} C_VEL
LIN {X 0,Y 573.259,Z 422.702,A -85,B 0,C 180,E1 -2311.968,E2 -2311.968} C_VEL
LIN {X 0,Y 573.254,Z 422.704,A -85,B 0,C 180,E1 -2314.59,E2 -2314.59} C_VEL
LIN {X 0,Y 573.233,Z 422.705,A -85,B 0,C 180,E1 -2317.662,E2 -2317.662} C_VEL
LIN {X 0,Y 573.251,Z 422.706,A -85,B 0,C 180,E1 -2319.923,E2 -2319.923} C_VEL
LIN {X 0,Y 573.256,Z 422.703,A -85,B 0,C 180,E1 -2322.988,E2 -2322.988} C_VEL
LIN {X 0,Y 573.266,Z 422.701,A -85,B 0,C 180,E1 -2325.807,E2 -2325.807} C_VEL
LIN {X 0,Y 573.276,Z 422.7,A -85,B 0,C 180,E1 -2328.734,E2 -2328.734} C_VEL
LIN {X 0,Y 573.302,Z 422.697,A -85,B 0,C 180,E1 -2331.541,E2 -2331.541} C_VEL
LIN {X 0,Y 573.289,Z 422.699,A -85,B 0,C 180,E1 -2334.372,E2 -2334.372} C_VEL
LIN {X 0,Y 573.303,Z 422.698,A -85,B 0,C 180,E1 -2337.893,E2 -2337.893} C_VEL
LIN {X 0,Y 573.329,Z 422.695,A -85,B 0,C 180,E1 -2340.703,E2 -2340.703} C_VEL
LIN {X 0,Y 573.238,Z 422.705,A -85,B 0,C 180,E1 -2343.515,E2 -2343.515} C_VEL
LIN {X 0,Y 573.298,Z 422.699,A -85,B 0,C 180,E1 -2345.628,E2 -2345.628} C_VEL
LIN {X 0,Y 573.301,Z 422.7,A -85,B 0,C 180,E1 -2348.459,E2 -2348.459} C_VEL
LIN {X 0,Y 573.264,Z 422.706,A -85,B 0,C 180,E1 -2351.312,E2 -2351.312} C_VEL
LIN {X 0,Y 573.267,Z 422.705,A -85,B 0,C 180,E1 -2354.193,E2 -2354.193} C_VEL
LIN {X 0,Y 573.255,Z 422.704,A -85,B 0,C 180,E1 -2357.112,E2 -2357.112} C_VEL
LIN {X 0,Y 573.252,Z 422.704,A -85,B 0,C 180,E1 -2360.077,E2 -2360.077} C_VEL
